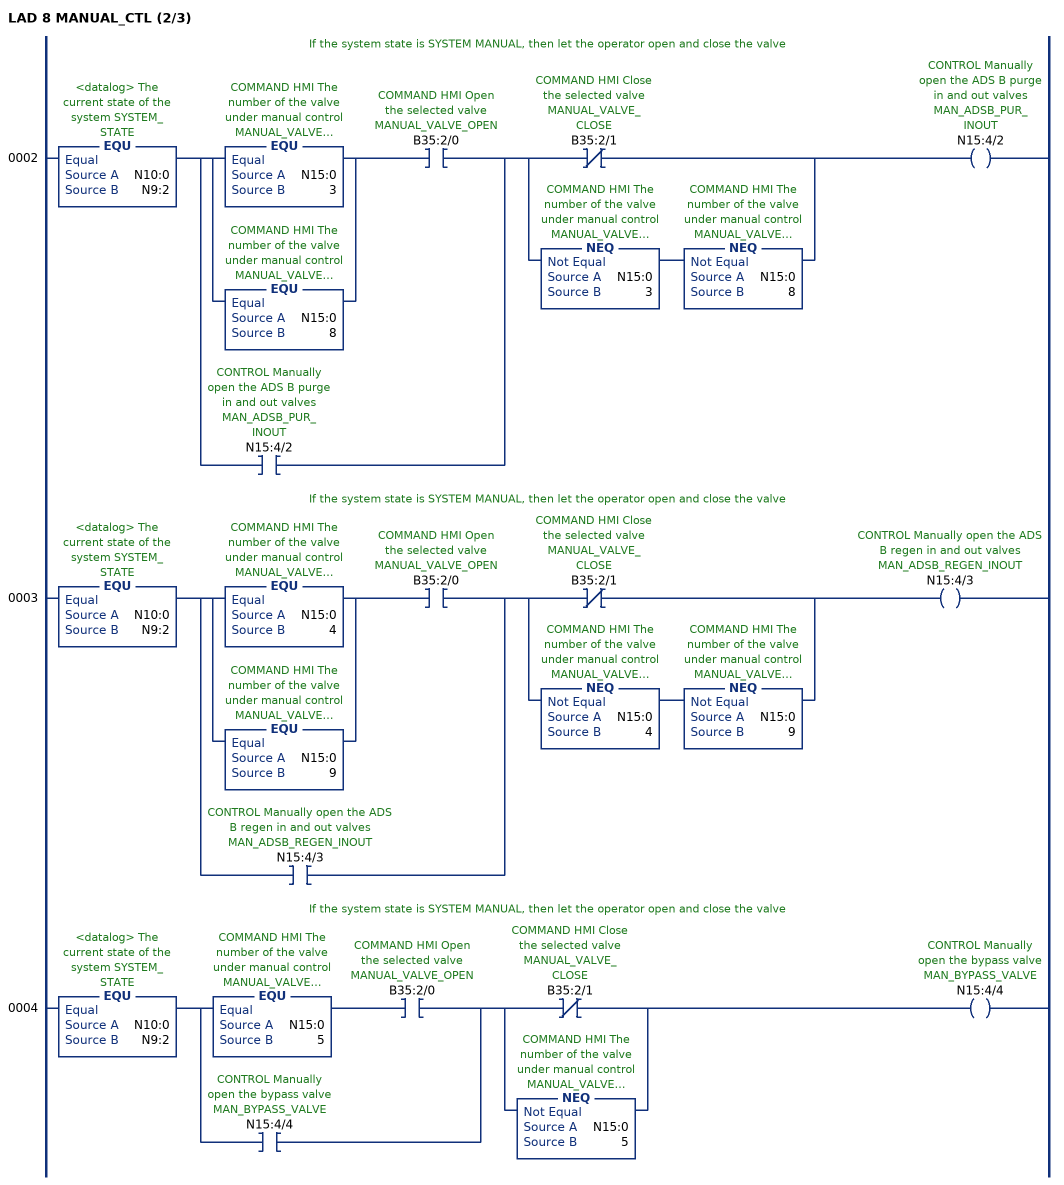
% Rung: 2 %
% If the system state is SYSTEM MANUAL, then let the operator open and close the valve %
SOR EQU N10:0 N9:2 BST BST EQU N15:0 3 NXB EQU N15:0 8 BND XIC B35:2/0 NXB XIC N15:4/2 BND BST XIO B35:2/1 NXB NEQ N15:0 3 NEQ N15:0 8 BND OTE N15:4/2 EOR
%   N10:0  SYSTEM_STATE  "<datalog> The current state of the system" %
%   N9:2  SYSTEM_MANUAL  "STATE System Manual" %
%   N15:0  MANUAL_VALVE_NUMBER  "COMMAND HMI The number of the valve under manual control" %
%   B35:2/0  MANUAL_VALVE_OPEN  "COMMAND HMI Open the selected valve" %
%   N15:4/2  MAN_ADSB_PUR_INOUT  "CONTROL Manually open the ADS B purge in and out valves" %
%   B35:2/1  MANUAL_VALVE_CLOSE  "COMMAND HMI Close the selected valve" %
% Rung: 3 %
% If the system state is SYSTEM MANUAL, then let the operator open and close the valve %
SOR EQU N10:0 N9:2 BST BST EQU N15:0 4 NXB EQU N15:0 9 BND XIC B35:2/0 NXB XIC N15:4/3 BND BST XIO B35:2/1 NXB NEQ N15:0 4 NEQ N15:0 9 BND OTE N15:4/3 EOR
%   N10:0  SYSTEM_STATE  "<datalog> The current state of the system" %
%   N9:2  SYSTEM_MANUAL  "STATE System Manual" %
%   N15:0  MANUAL_VALVE_NUMBER  "COMMAND HMI The number of the valve under manual control" %
%   B35:2/0  MANUAL_VALVE_OPEN  "COMMAND HMI Open the selected valve" %
%   N15:4/3  MAN_ADSB_REGEN_INOUT  "CONTROL Manually open the ADS B regen in and out valves" %
%   B35:2/1  MANUAL_VALVE_CLOSE  "COMMAND HMI Close the selected valve" %
% Rung: 4 %
% If the system state is SYSTEM MANUAL, then let the operator open and close the valve %
SOR EQU N10:0 N9:2 BST EQU N15:0 5 XIC B35:2/0 NXB XIC N15:4/4 BND BST XIO B35:2/1 NXB NEQ N15:0 5 BND OTE N15:4/4 EOR
%   N10:0  SYSTEM_STATE  "<datalog> The current state of the system" %
%   N9:2  SYSTEM_MANUAL  "STATE System Manual" %
%   N15:0  MANUAL_VALVE_NUMBER  "COMMAND HMI The number of the valve under manual control" %
%   B35:2/0  MANUAL_VALVE_OPEN  "COMMAND HMI Open the selected valve" %
%   N15:4/4  MAN_BYPASS_VALVE  "CONTROL Manually open the bypass valve" %
%   B35:2/1  MANUAL_VALVE_CLOSE  "COMMAND HMI Close the selected valve" %

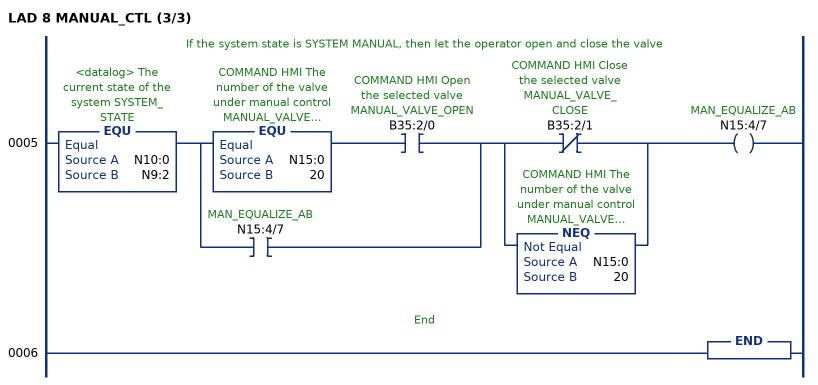
% Rung: 5 %
% If the system state is SYSTEM MANUAL, then let the operator open and close the valve %
SOR EQU N10:0 N9:2 BST EQU N15:0 20 XIC B35:2/0 NXB XIC N15:4/7 BND BST XIO B35:2/1 NXB NEQ N15:0 20 BND OTE N15:4/7 EOR
%   N10:0  SYSTEM_STATE  "<datalog> The current state of the system" %
%   N9:2  SYSTEM_MANUAL  "STATE System Manual" %
%   N15:0  MANUAL_VALVE_NUMBER  "COMMAND HMI The number of the valve under manual control" %
%   B35:2/0  MANUAL_VALVE_OPEN  "COMMAND HMI Open the selected valve" %
%   N15:4/7  MAN_EQUALIZE_AB %
%   B35:2/1  MANUAL_VALVE_CLOSE  "COMMAND HMI Close the selected valve" %
% Rung: 6 %
% End %
SOR END EOR

LADDER 10 "PURIFY"    % Operates the purify control %
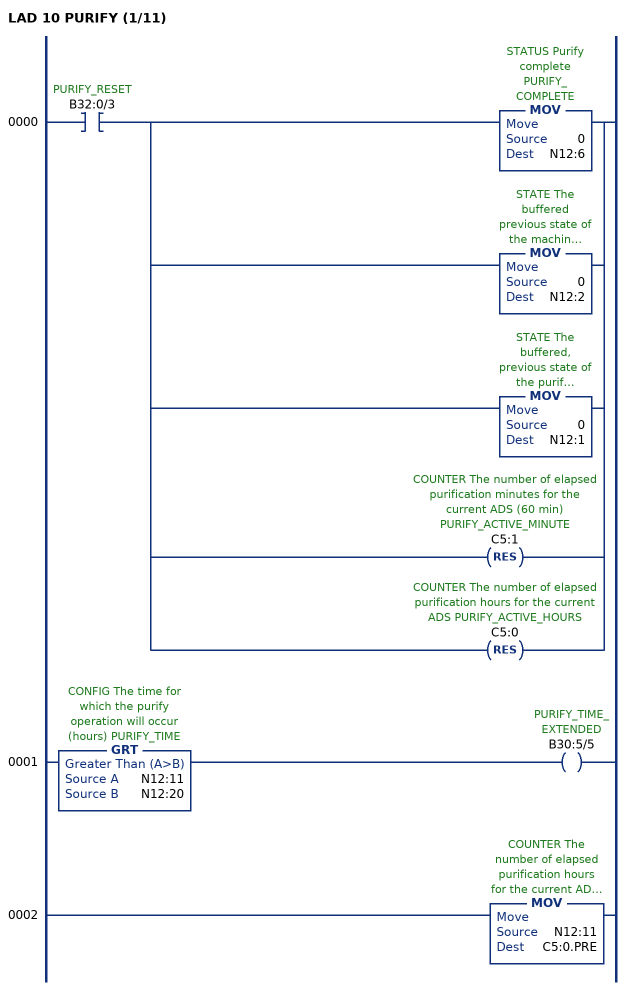
% Rung: 0 %
SOR XIC B32:0/3 BST MOV 0 N12:6 NXB MOV 0 N12:2 NXB MOV 0 N12:1 NXB RES C5:1 NXB RES C5:0 BND EOR
%   B32:0/3  PURIFY_RESET %
%   N12:6  PURIFY_COMPLETE  "STATUS Purify complete" %
%   N12:2  PURIFY_ALARM_BUFFER  "STATE The buffered previous state of the machine when the system alarm occured" %
%   N12:1  PURIFY_STDBY_BUFFER  "STATE The buffered, previous state of the purify process" %
%   C5:1  PURIFY_ACTIVE_MINUTE  "COUNTER The number of elapsed purification minutes for the current ADS (60 min)" %
%   C5:0  PURIFY_ACTIVE_HOURS  "COUNTER The number of elapsed purification hours for the current ADS" %
% Rung: 1 %
SOR GRT N12:11 N12:20 OTE B30:5/5 EOR
%   N12:11  PURIFY_TIME  "CONFIG The time for which the purify operation will occur (hours)" %
%   N12:20  DEFAULT_PURIFY_TIME %
%   B30:5/5  PURIFY_TIME_EXTENDED %
% Rung: 2 %
SOR MOV N12:11 C5:0.PRE EOR
%   N12:11  PURIFY_TIME  "CONFIG The time for which the purify operation will occur (hours)" %
%   C5:0  PURIFY_ACTIVE_HOURS  "COUNTER The number of elapsed purification hours for the current ADS" %

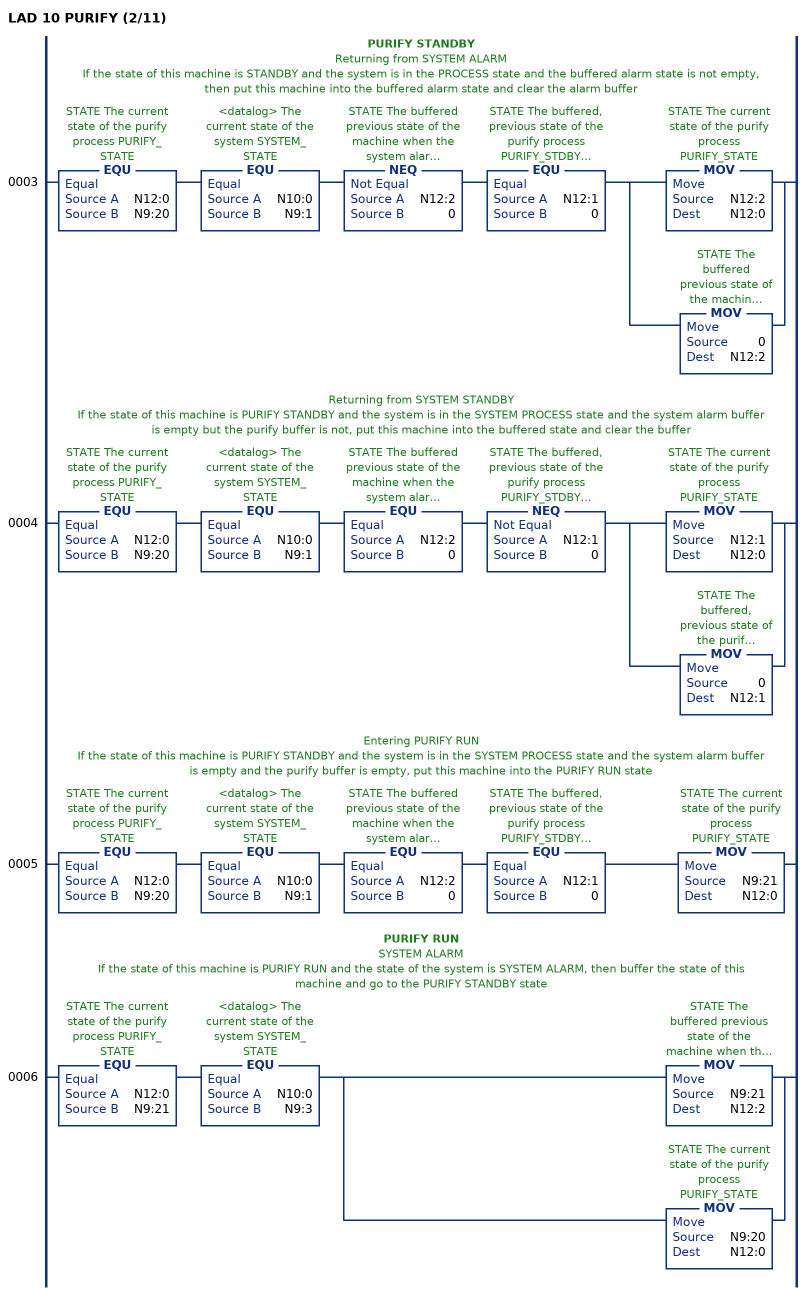
% Rung: 3 %
% TITLE: PURIFY STANDBY %
% Returning from SYSTEM ALARM
% If the state of this machine is STANDBY and the system is in the PROCESS state and the buffered alarm state is not empty, then put this machine into the buffered alarm state and clear the alarm buffer %
SOR EQU N12:0 N9:20 EQU N10:0 N9:1 NEQ N12:2 0 EQU N12:1 0 BST MOV N12:2 N12:0 NXB MOV 0 N12:2 BND EOR
%   N12:0  PURIFY_STATE  "STATE The current state of the purify process" %
%   N9:20  PURIFY_STANDBY  "STATE Purify Standby" %
%   N10:0  SYSTEM_STATE  "<datalog> The current state of the system" %
%   N9:1  SYSTEM_PROCESS  "STATE System Process" %
%   N12:2  PURIFY_ALARM_BUFFER  "STATE The buffered previous state of the machine when the system alarm occured" %
%   N12:1  PURIFY_STDBY_BUFFER  "STATE The buffered, previous state of the purify process" %
% Rung: 4 %
% Returning from SYSTEM STANDBY
% If the state of this machine is PURIFY STANDBY and the system is in the SYSTEM PROCESS state and the system alarm buffer is empty but the purify buffer is not, put this machine into the buffered state and clear the buffer %
SOR EQU N12:0 N9:20 EQU N10:0 N9:1 EQU N12:2 0 NEQ N12:1 0 BST MOV N12:1 N12:0 NXB MOV 0 N12:1 BND EOR
%   N12:0  PURIFY_STATE  "STATE The current state of the purify process" %
%   N9:20  PURIFY_STANDBY  "STATE Purify Standby" %
%   N10:0  SYSTEM_STATE  "<datalog> The current state of the system" %
%   N9:1  SYSTEM_PROCESS  "STATE System Process" %
%   N12:2  PURIFY_ALARM_BUFFER  "STATE The buffered previous state of the machine when the system alarm occured" %
%   N12:1  PURIFY_STDBY_BUFFER  "STATE The buffered, previous state of the purify process" %
% Rung: 5 %
% Entering PURIFY RUN
% If the state of this machine is PURIFY STANDBY and the system is in the SYSTEM PROCESS state and the system alarm buffer is empty and the purify buffer is empty, put this machine into the PURIFY RUN state %
SOR EQU N12:0 N9:20 EQU N10:0 N9:1 EQU N12:2 0 EQU N12:1 0 MOV N9:21 N12:0 EOR
%   N12:0  PURIFY_STATE  "STATE The current state of the purify process" %
%   N9:20  PURIFY_STANDBY  "STATE Purify Standby" %
%   N10:0  SYSTEM_STATE  "<datalog> The current state of the system" %
%   N9:1  SYSTEM_PROCESS  "STATE System Process" %
%   N12:2  PURIFY_ALARM_BUFFER  "STATE The buffered previous state of the machine when the system alarm occured" %
%   N12:1  PURIFY_STDBY_BUFFER  "STATE The buffered, previous state of the purify process" %
%   N9:21  PURIFY_RUN  "STATE Purify running" %
% Rung: 6 %
% TITLE: PURIFY RUN %
% SYSTEM ALARM
% If the state of this machine is PURIFY RUN and the state of the system is SYSTEM ALARM, then buffer the state of this machine and go to the PURIFY STANDBY state %
SOR EQU N12:0 N9:21 EQU N10:0 N9:3 BST MOV N9:21 N12:2 NXB MOV N9:20 N12:0 BND EOR
%   N12:0  PURIFY_STATE  "STATE The current state of the purify process" %
%   N9:21  PURIFY_RUN  "STATE Purify running" %
%   N10:0  SYSTEM_STATE  "<datalog> The current state of the system" %
%   N9:3  SYSTEM_ALARM  "STATE System Alarm" %
%   N12:2  PURIFY_ALARM_BUFFER  "STATE The buffered previous state of the machine when the system alarm occured" %
%   N9:20  PURIFY_STANDBY  "STATE Purify Standby" %

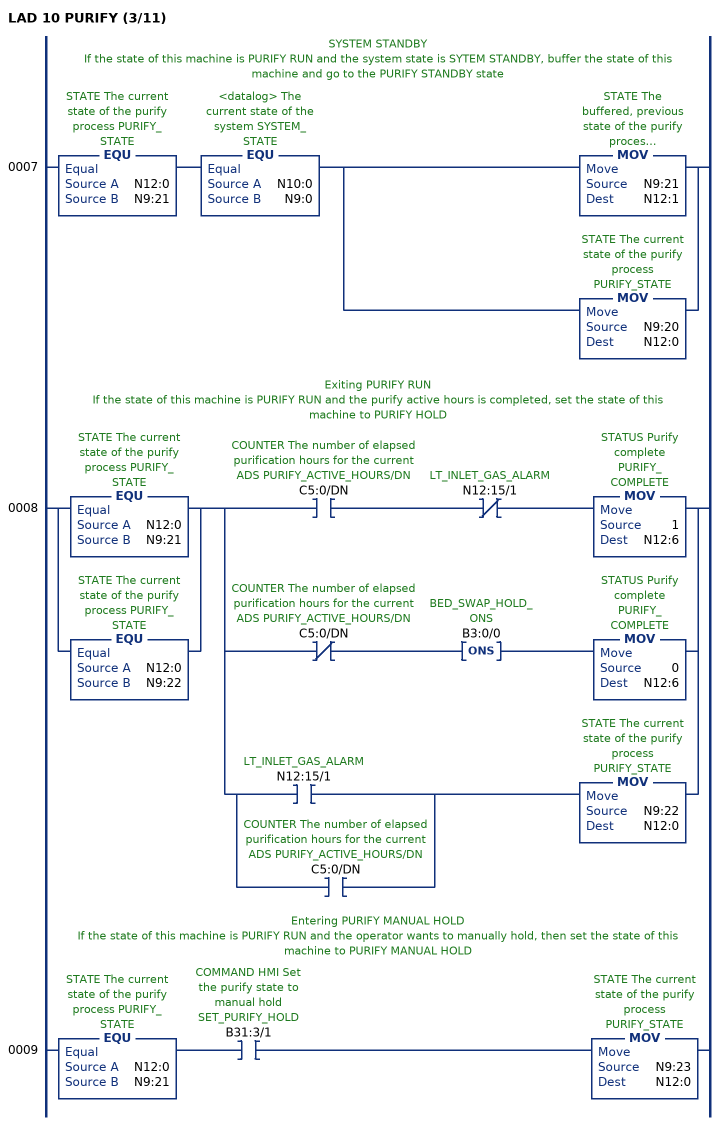
% Rung: 7 %
% SYSTEM STANDBY
% If the state of this machine is PURIFY RUN and the system state is SYTEM STANDBY, buffer the state of this machine and go to the PURIFY STANDBY state %
SOR EQU N12:0 N9:21 EQU N10:0 N9:0 BST MOV N9:21 N12:1 NXB MOV N9:20 N12:0 BND EOR
%   N12:0  PURIFY_STATE  "STATE The current state of the purify process" %
%   N9:21  PURIFY_RUN  "STATE Purify running" %
%   N10:0  SYSTEM_STATE  "<datalog> The current state of the system" %
%   N9:0  SYSTEM_STANDBY  "STATE System Standby" %
%   N12:1  PURIFY_STDBY_BUFFER  "STATE The buffered, previous state of the purify process" %
%   N9:20  PURIFY_STANDBY  "STATE Purify Standby" %
% Rung: 8 %
% Exiting PURIFY RUN
% If the state of this machine is PURIFY RUN and the purify active hours is completed, set the state of this machine to PURIFY HOLD %
SOR BST EQU N12:0 N9:21 NXB EQU N12:0 N9:22 BND BST XIC C5:0/DN XIO N12:15/1 MOV 1 N12:6 NXB XIO C5:0/DN ONS B3:0/0 MOV 0 N12:6 NXB BST XIC N12:15/1 NXB XIC C5:0/DN BND MOV N9:22 N12:0 BND EOR
%   N12:0  PURIFY_STATE  "STATE The current state of the purify process" %
%   N9:21  PURIFY_RUN  "STATE Purify running" %
%   N9:22  PURIFY_HOLD  "STATE Purify Hold" %
%   C5:0  PURIFY_ACTIVE_HOURS  "COUNTER The number of elapsed purification hours for the current ADS" %
%   N12:15/1  LT_INLET_GAS_ALARM %
%   N12:6  PURIFY_COMPLETE  "STATUS Purify complete" %
%   B3:0/0  BED_SWAP_HOLD_ONS %
% Rung: 9 %
% Entering PURIFY MANUAL HOLD
% If the state of this machine is PURIFY RUN and the operator wants to manually hold, then set the state of this machine to PURIFY MANUAL HOLD %
SOR EQU N12:0 N9:21 XIC B31:3/1 MOV N9:23 N12:0 EOR
%   N12:0  PURIFY_STATE  "STATE The current state of the purify process" %
%   N9:21  PURIFY_RUN  "STATE Purify running" %
%   B31:3/1  SET_PURIFY_HOLD  "COMMAND HMI Set the purify state to manual hold" %
%   N9:23  PURIFY_MANUAL_HOLD  "STATE Purify Manual Hold" %

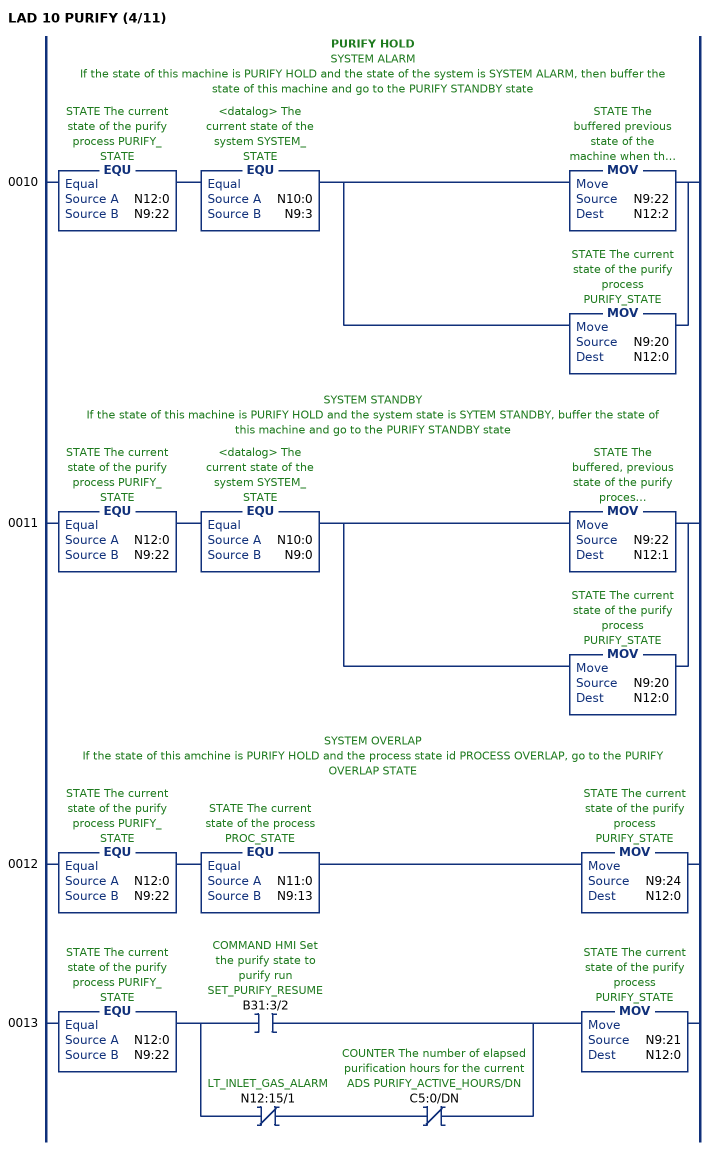
% Rung: 10 %
% TITLE: PURIFY HOLD %
% SYSTEM ALARM
% If the state of this machine is PURIFY HOLD and the state of the system is SYSTEM ALARM, then buffer the state of this machine and go to the PURIFY STANDBY state %
SOR EQU N12:0 N9:22 EQU N10:0 N9:3 BST MOV N9:22 N12:2 NXB MOV N9:20 N12:0 BND EOR
%   N12:0  PURIFY_STATE  "STATE The current state of the purify process" %
%   N9:22  PURIFY_HOLD  "STATE Purify Hold" %
%   N10:0  SYSTEM_STATE  "<datalog> The current state of the system" %
%   N9:3  SYSTEM_ALARM  "STATE System Alarm" %
%   N12:2  PURIFY_ALARM_BUFFER  "STATE The buffered previous state of the machine when the system alarm occured" %
%   N9:20  PURIFY_STANDBY  "STATE Purify Standby" %
% Rung: 11 %
% SYSTEM STANDBY
% If the state of this machine is PURIFY HOLD and the system state is SYTEM STANDBY, buffer the state of this machine and go to the PURIFY STANDBY state %
SOR EQU N12:0 N9:22 EQU N10:0 N9:0 BST MOV N9:22 N12:1 NXB MOV N9:20 N12:0 BND EOR
%   N12:0  PURIFY_STATE  "STATE The current state of the purify process" %
%   N9:22  PURIFY_HOLD  "STATE Purify Hold" %
%   N10:0  SYSTEM_STATE  "<datalog> The current state of the system" %
%   N9:0  SYSTEM_STANDBY  "STATE System Standby" %
%   N12:1  PURIFY_STDBY_BUFFER  "STATE The buffered, previous state of the purify process" %
%   N9:20  PURIFY_STANDBY  "STATE Purify Standby" %
% Rung: 12 %
% SYSTEM OVERLAP
% If the state of this amchine is PURIFY HOLD and the process state id PROCESS OVERLAP, go to the PURIFY OVERLAP STATE %
SOR EQU N12:0 N9:22 EQU N11:0 N9:13 MOV N9:24 N12:0 EOR
%   N12:0  PURIFY_STATE  "STATE The current state of the purify process" %
%   N9:22  PURIFY_HOLD  "STATE Purify Hold" %
%   N11:0  PROC_STATE  "STATE The current state of the process" %
%   N9:13  PROC_OVERLAP  "STATE Process Purify Overlap" %
%   N9:24  PURIFY_OVERLAP  "STATE Puriify Overlap" %
% Rung: 13 %
SOR EQU N12:0 N9:22 BST XIC B31:3/2 NXB XIO N12:15/1 XIO C5:0/DN BND MOV N9:21 N12:0 EOR
%   N12:0  PURIFY_STATE  "STATE The current state of the purify process" %
%   N9:22  PURIFY_HOLD  "STATE Purify Hold" %
%   B31:3/2  SET_PURIFY_RESUME  "COMMAND HMI Set the purify state to purify run" %
%   N12:15/1  LT_INLET_GAS_ALARM %
%   C5:0  PURIFY_ACTIVE_HOURS  "COUNTER The number of elapsed purification hours for the current ADS" %
%   N9:21  PURIFY_RUN  "STATE Purify running" %

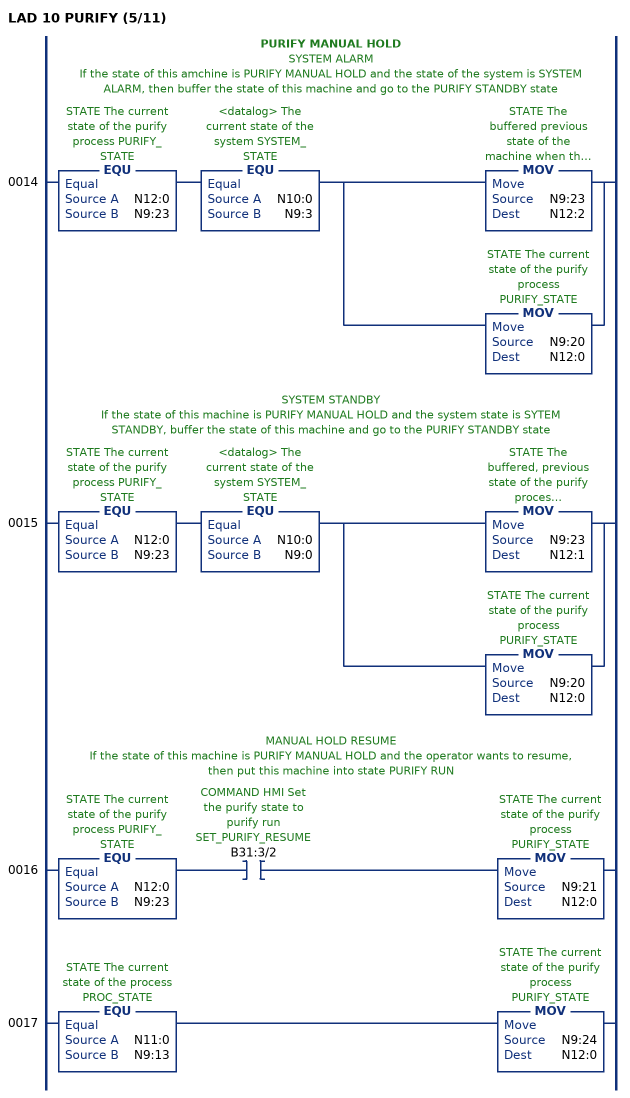
% Rung: 14 %
% TITLE: PURIFY MANUAL HOLD %
% SYSTEM ALARM
% If the state of this amchine is PURIFY MANUAL HOLD and the state of the system is SYSTEM ALARM, then buffer the state of this machine and go to the PURIFY STANDBY state %
SOR EQU N12:0 N9:23 EQU N10:0 N9:3 BST MOV N9:23 N12:2 NXB MOV N9:20 N12:0 BND EOR
%   N12:0  PURIFY_STATE  "STATE The current state of the purify process" %
%   N9:23  PURIFY_MANUAL_HOLD  "STATE Purify Manual Hold" %
%   N10:0  SYSTEM_STATE  "<datalog> The current state of the system" %
%   N9:3  SYSTEM_ALARM  "STATE System Alarm" %
%   N12:2  PURIFY_ALARM_BUFFER  "STATE The buffered previous state of the machine when the system alarm occured" %
%   N9:20  PURIFY_STANDBY  "STATE Purify Standby" %
% Rung: 15 %
% SYSTEM STANDBY
% If the state of this machine is PURIFY MANUAL HOLD and the system state is SYTEM STANDBY, buffer the state of this machine and go to the PURIFY STANDBY state %
SOR EQU N12:0 N9:23 EQU N10:0 N9:0 BST MOV N9:23 N12:1 NXB MOV N9:20 N12:0 BND EOR
%   N12:0  PURIFY_STATE  "STATE The current state of the purify process" %
%   N9:23  PURIFY_MANUAL_HOLD  "STATE Purify Manual Hold" %
%   N10:0  SYSTEM_STATE  "<datalog> The current state of the system" %
%   N9:0  SYSTEM_STANDBY  "STATE System Standby" %
%   N12:1  PURIFY_STDBY_BUFFER  "STATE The buffered, previous state of the purify process" %
%   N9:20  PURIFY_STANDBY  "STATE Purify Standby" %
% Rung: 16 %
% MANUAL HOLD RESUME
% If the state of this machine is PURIFY MANUAL HOLD and the operator wants to resume, then put this machine into state PURIFY RUN %
SOR EQU N12:0 N9:23 XIC B31:3/2 MOV N9:21 N12:0 EOR
%   N12:0  PURIFY_STATE  "STATE The current state of the purify process" %
%   N9:23  PURIFY_MANUAL_HOLD  "STATE Purify Manual Hold" %
%   B31:3/2  SET_PURIFY_RESUME  "COMMAND HMI Set the purify state to purify run" %
%   N9:21  PURIFY_RUN  "STATE Purify running" %
% Rung: 17 %
SOR EQU N11:0 N9:13 MOV N9:24 N12:0 EOR
%   N11:0  PROC_STATE  "STATE The current state of the process" %
%   N9:13  PROC_OVERLAP  "STATE Process Purify Overlap" %
%   N9:24  PURIFY_OVERLAP  "STATE Puriify Overlap" %
%   N12:0  PURIFY_STATE  "STATE The current state of the purify process" %

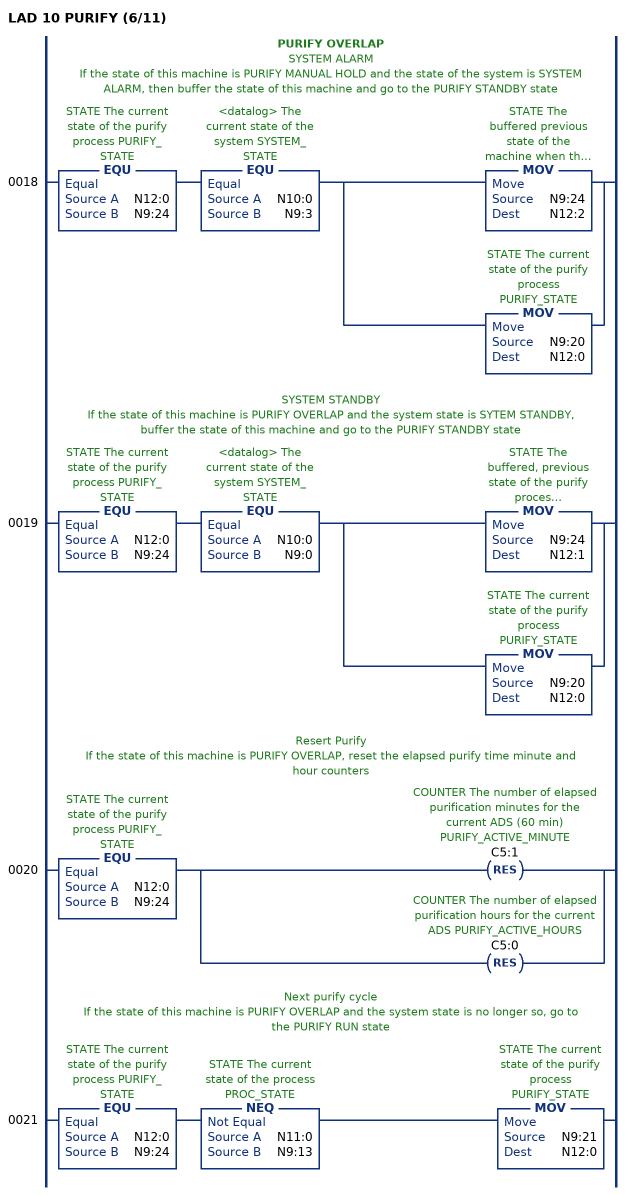
% Rung: 18 %
% TITLE: PURIFY OVERLAP %
% SYSTEM ALARM
% If the state of this machine is PURIFY MANUAL HOLD and the state of the system is SYSTEM ALARM, then buffer the state of this machine and go to the PURIFY STANDBY state %
SOR EQU N12:0 N9:24 EQU N10:0 N9:3 BST MOV N9:24 N12:2 NXB MOV N9:20 N12:0 BND EOR
%   N12:0  PURIFY_STATE  "STATE The current state of the purify process" %
%   N9:24  PURIFY_OVERLAP  "STATE Puriify Overlap" %
%   N10:0  SYSTEM_STATE  "<datalog> The current state of the system" %
%   N9:3  SYSTEM_ALARM  "STATE System Alarm" %
%   N12:2  PURIFY_ALARM_BUFFER  "STATE The buffered previous state of the machine when the system alarm occured" %
%   N9:20  PURIFY_STANDBY  "STATE Purify Standby" %
% Rung: 19 %
% SYSTEM STANDBY
% If the state of this machine is PURIFY OVERLAP and the system state is SYTEM STANDBY, buffer the state of this machine and go to the PURIFY STANDBY state %
SOR EQU N12:0 N9:24 EQU N10:0 N9:0 BST MOV N9:24 N12:1 NXB MOV N9:20 N12:0 BND EOR
%   N12:0  PURIFY_STATE  "STATE The current state of the purify process" %
%   N9:24  PURIFY_OVERLAP  "STATE Puriify Overlap" %
%   N10:0  SYSTEM_STATE  "<datalog> The current state of the system" %
%   N9:0  SYSTEM_STANDBY  "STATE System Standby" %
%   N12:1  PURIFY_STDBY_BUFFER  "STATE The buffered, previous state of the purify process" %
%   N9:20  PURIFY_STANDBY  "STATE Purify Standby" %
% Rung: 20 %
% Resert Purify
% If the state of this machine is PURIFY OVERLAP, reset the elapsed purify time minute and hour counters %
SOR EQU N12:0 N9:24 BST RES C5:1 NXB RES C5:0 BND EOR
%   N12:0  PURIFY_STATE  "STATE The current state of the purify process" %
%   N9:24  PURIFY_OVERLAP  "STATE Puriify Overlap" %
%   C5:1  PURIFY_ACTIVE_MINUTE  "COUNTER The number of elapsed purification minutes for the current ADS (60 min)" %
%   C5:0  PURIFY_ACTIVE_HOURS  "COUNTER The number of elapsed purification hours for the current ADS" %
% Rung: 21 %
% Next purify cycle
% If the state of this machine is PURIFY OVERLAP and the system state is no longer so, go to the PURIFY RUN state %
SOR EQU N12:0 N9:24 NEQ N11:0 N9:13 MOV N9:21 N12:0 EOR
%   N12:0  PURIFY_STATE  "STATE The current state of the purify process" %
%   N9:24  PURIFY_OVERLAP  "STATE Puriify Overlap" %
%   N11:0  PROC_STATE  "STATE The current state of the process" %
%   N9:13  PROC_OVERLAP  "STATE Process Purify Overlap" %
%   N9:21  PURIFY_RUN  "STATE Purify running" %

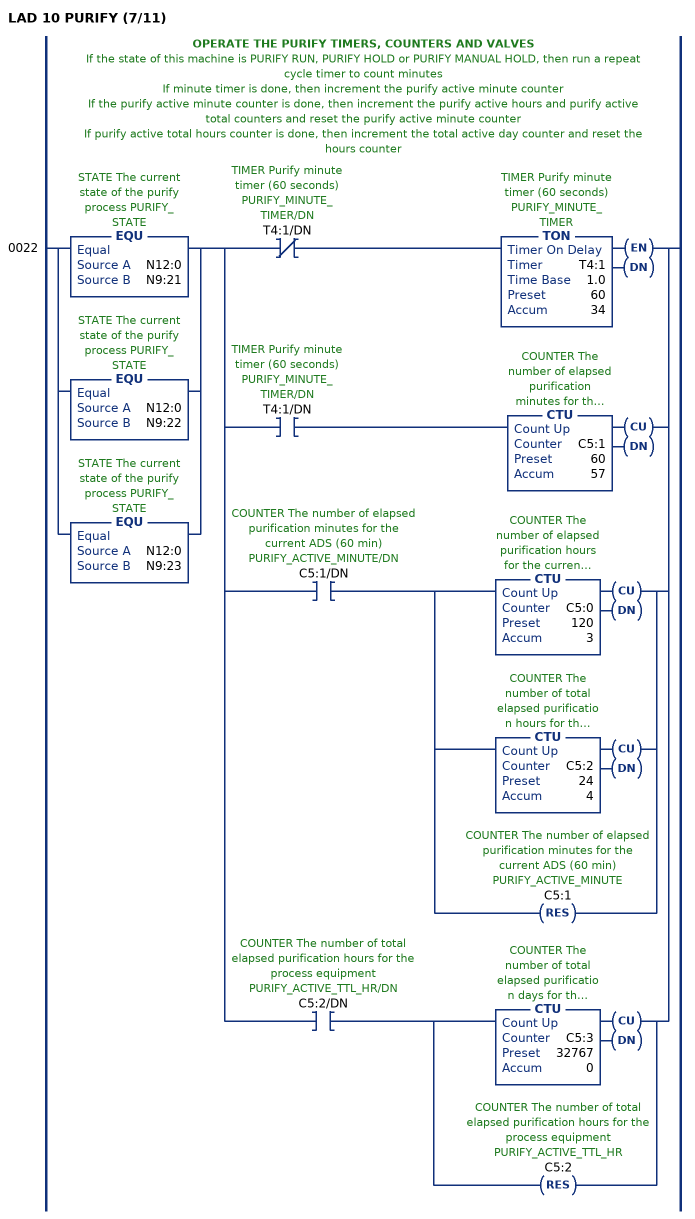
% Rung: 22 %
% TITLE: OPERATE THE PURIFY TIMERS, COUNTERS AND VALVES %
% If the state of this machine is PURIFY RUN, PURIFY HOLD or PURIFY MANUAL HOLD, then run a repeat cycle timer to count minutes
% If minute timer is done, then increment the purify active minute counter
% If the purify active minute counter is done, then increment the purify active hours and purify active total counters and reset the purify active minute counter
% If purify active total hours counter is done, then increment the total active day counter and reset the hours counter %
SOR BST EQU N12:0 N9:21 NXB EQU N12:0 N9:22 NXB EQU N12:0 N9:23 BND BST XIO T4:1/DN TON T4:1 1.0 60 34 NXB XIC T4:1/DN CTU C5:1 60 57 NXB XIC C5:1/DN BST CTU C5:0 120 3 NXB CTU C5:2 24 4 NXB RES C5:1 BND NXB XIC C5:2/DN BST CTU C5:3 32767 0 NXB RES C5:2 BND BND EOR
%   N12:0  PURIFY_STATE  "STATE The current state of the purify process" %
%   N9:21  PURIFY_RUN  "STATE Purify running" %
%   N9:22  PURIFY_HOLD  "STATE Purify Hold" %
%   N9:23  PURIFY_MANUAL_HOLD  "STATE Purify Manual Hold" %
%   T4:1  PURIFY_MINUTE_TIMER  "TIMER Purify minute timer (60 seconds)" %
%   C5:1  PURIFY_ACTIVE_MINUTE  "COUNTER The number of elapsed purification minutes for the current ADS (60 min)" %
%   C5:0  PURIFY_ACTIVE_HOURS  "COUNTER The number of elapsed purification hours for the current ADS" %
%   C5:2  PURIFY_ACTIVE_TTL_HR  "COUNTER The number of total elapsed purification hours for the process equipment" %
%   C5:3  PURIFY_ACTIVE_TTL_DY  "COUNTER The number of total elapsed purification days for the process equipment" %

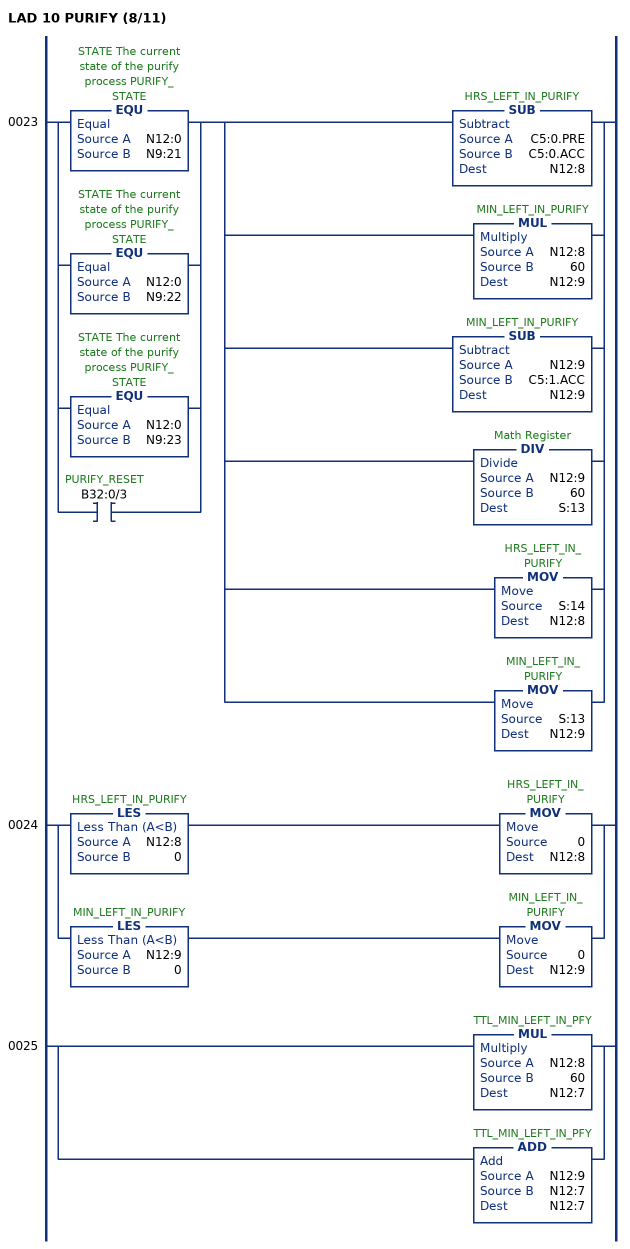
% Rung: 23 %
SOR BST EQU N12:0 N9:21 NXB EQU N12:0 N9:22 NXB EQU N12:0 N9:23 NXB XIC B32:0/3 BND BST SUB C5:0.PRE C5:0.ACC N12:8 NXB MUL N12:8 60 N12:9 NXB SUB N12:9 C5:1.ACC N12:9 NXB DIV N12:9 60 S:13 NXB MOV S:14 N12:8 NXB MOV S:13 N12:9 BND EOR
%   N12:0  PURIFY_STATE  "STATE The current state of the purify process" %
%   N9:21  PURIFY_RUN  "STATE Purify running" %
%   N9:22  PURIFY_HOLD  "STATE Purify Hold" %
%   N9:23  PURIFY_MANUAL_HOLD  "STATE Purify Manual Hold" %
%   B32:0/3  PURIFY_RESET %
%   C5:0  PURIFY_ACTIVE_HOURS  "COUNTER The number of elapsed purification hours for the current ADS" %
%   N12:8  HRS_LEFT_IN_PURIFY %
%   N12:9  MIN_LEFT_IN_PURIFY %
%   C5:1  PURIFY_ACTIVE_MINUTE  "COUNTER The number of elapsed purification minutes for the current ADS (60 min)" %
%   S:13  "Math Register" %
%   S:14  "Math Register" %
% Rung: 24 %
SOR BST LES N12:8 0 MOV 0 N12:8 NXB LES N12:9 0 MOV 0 N12:9 BND EOR
%   N12:8  HRS_LEFT_IN_PURIFY %
%   N12:9  MIN_LEFT_IN_PURIFY %
% Rung: 25 %
SOR BST MUL N12:8 60 N12:7 NXB ADD N12:9 N12:7 N12:7 BND EOR
%   N12:8  HRS_LEFT_IN_PURIFY %
%   N12:7  TTL_MIN_LEFT_IN_PFY %
%   N12:9  MIN_LEFT_IN_PURIFY %

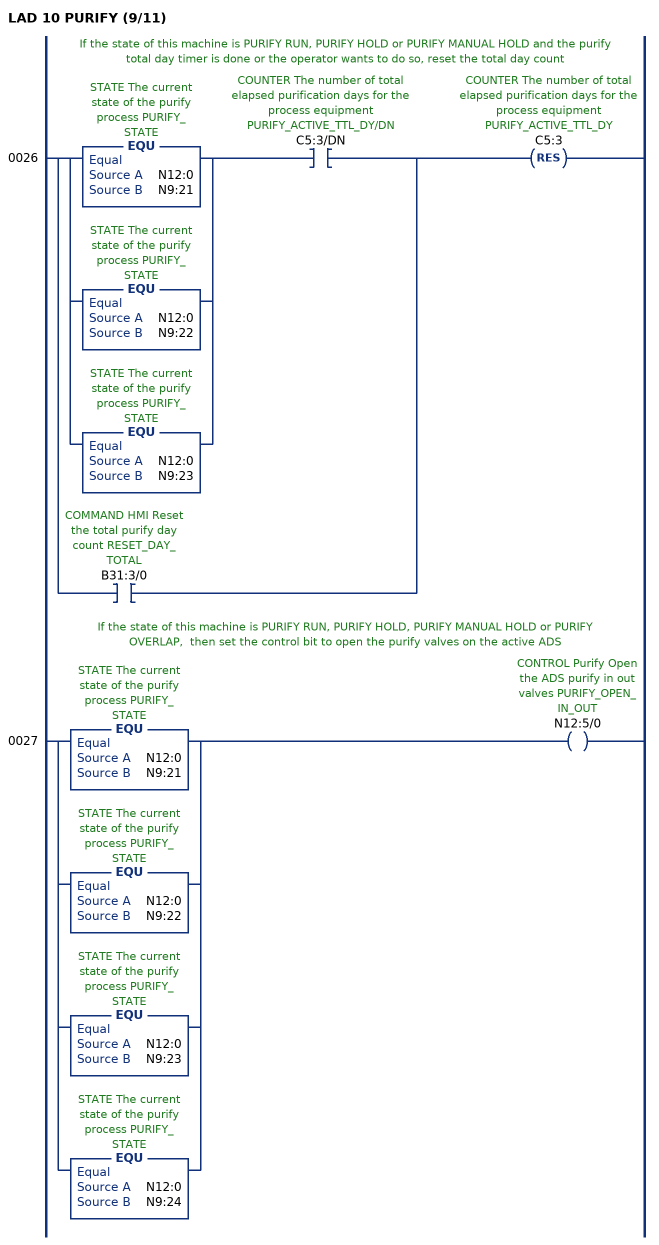
% Rung: 26 %
% If the state of this machine is PURIFY RUN, PURIFY HOLD or PURIFY MANUAL HOLD and the purify total day timer is done or the operator wants to do so, reset the total day count %
SOR BST BST EQU N12:0 N9:21 NXB EQU N12:0 N9:22 NXB EQU N12:0 N9:23 BND XIC C5:3/DN NXB XIC B31:3/0 BND RES C5:3 EOR
%   N12:0  PURIFY_STATE  "STATE The current state of the purify process" %
%   N9:21  PURIFY_RUN  "STATE Purify running" %
%   N9:22  PURIFY_HOLD  "STATE Purify Hold" %
%   N9:23  PURIFY_MANUAL_HOLD  "STATE Purify Manual Hold" %
%   C5:3  PURIFY_ACTIVE_TTL_DY  "COUNTER The number of total elapsed purification days for the process equipment" %
%   B31:3/0  RESET_DAY_TOTAL  "COMMAND HMI Reset the total purify day count" %
% Rung: 27 %
% If the state of this machine is PURIFY RUN, PURIFY HOLD, PURIFY MANUAL HOLD or PURIFY OVERLAP,  then set the control bit to open the purify valves on the active ADS %
SOR BST EQU N12:0 N9:21 NXB EQU N12:0 N9:22 NXB EQU N12:0 N9:23 NXB EQU N12:0 N9:24 BND OTE N12:5/0 EOR
%   N12:0  PURIFY_STATE  "STATE The current state of the purify process" %
%   N9:21  PURIFY_RUN  "STATE Purify running" %
%   N9:22  PURIFY_HOLD  "STATE Purify Hold" %
%   N9:23  PURIFY_MANUAL_HOLD  "STATE Purify Manual Hold" %
%   N9:24  PURIFY_OVERLAP  "STATE Puriify Overlap" %
%   N12:5/0  PURIFY_OPEN_IN_OUT  "CONTROL Purify Open the ADS purify in out valves" %

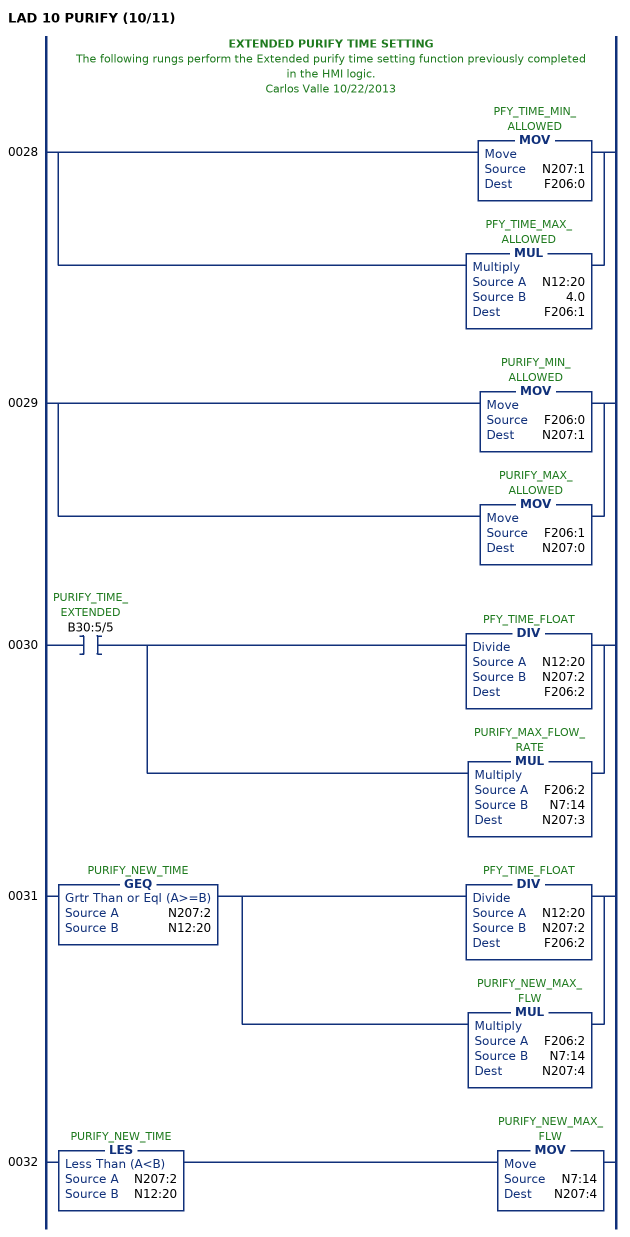
% Rung: 28 %
% TITLE: EXTENDED PURIFY TIME SETTING %
% The following rungs perform the Extended purify time setting function previously completed in the HMI logic.
% Carlos Valle 10/22/2013 %
SOR BST MOV N207:1 F206:0 NXB MUL N12:20 4.0 F206:1 BND EOR
%   N207:1  PURIFY_MIN_ALLOWED %
%   F206:0  PFY_TIME_MIN_ALLOWED %
%   N12:20  DEFAULT_PURIFY_TIME %
%   F206:1  PFY_TIME_MAX_ALLOWED %
% Rung: 29 %
SOR BST MOV F206:0 N207:1 NXB MOV F206:1 N207:0 BND EOR
%   F206:0  PFY_TIME_MIN_ALLOWED %
%   N207:1  PURIFY_MIN_ALLOWED %
%   F206:1  PFY_TIME_MAX_ALLOWED %
%   N207:0  PURIFY_MAX_ALLOWED %
% Rung: 30 %
SOR XIC B30:5/5 BST DIV N12:20 N207:2 F206:2 NXB MUL F206:2 N7:14 N207:3 BND EOR
%   B30:5/5  PURIFY_TIME_EXTENDED %
%   N12:20  DEFAULT_PURIFY_TIME %
%   N207:2  PURIFY_NEW_TIME %
%   F206:2  PFY_TIME_FLOAT %
%   N7:14  PURIFIER_SIZE %
%   N207:3  PURIFY_MAX_FLOW_RATE %
% Rung: 31 %
SOR GEQ N207:2 N12:20 BST DIV N12:20 N207:2 F206:2 NXB MUL F206:2 N7:14 N207:4 BND EOR
%   N207:2  PURIFY_NEW_TIME %
%   N12:20  DEFAULT_PURIFY_TIME %
%   F206:2  PFY_TIME_FLOAT %
%   N7:14  PURIFIER_SIZE %
%   N207:4  PURIFY_NEW_MAX_FLW %
% Rung: 32 %
SOR LES N207:2 N12:20 MOV N7:14 N207:4 EOR
%   N207:2  PURIFY_NEW_TIME %
%   N12:20  DEFAULT_PURIFY_TIME %
%   N7:14  PURIFIER_SIZE %
%   N207:4  PURIFY_NEW_MAX_FLW %

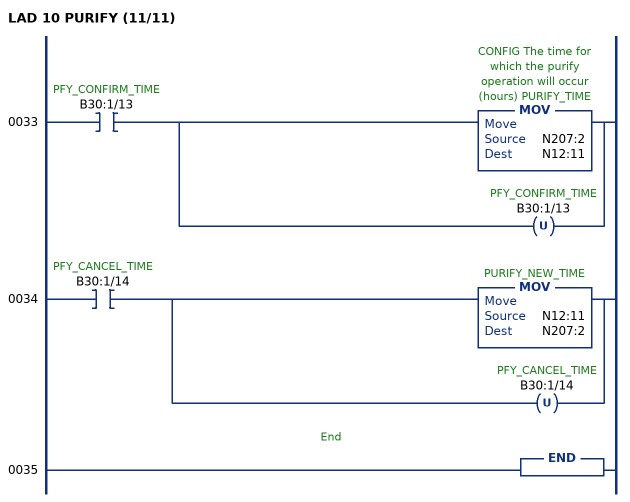
% Rung: 33 %
SOR XIC B30:1/13 BST MOV N207:2 N12:11 NXB OTU B30:1/13 BND EOR
%   B30:1/13  PFY_CONFIRM_TIME %
%   N207:2  PURIFY_NEW_TIME %
%   N12:11  PURIFY_TIME  "CONFIG The time for which the purify operation will occur (hours)" %
% Rung: 34 %
SOR XIC B30:1/14 BST MOV N12:11 N207:2 NXB OTU B30:1/14 BND EOR
%   B30:1/14  PFY_CANCEL_TIME %
%   N12:11  PURIFY_TIME  "CONFIG The time for which the purify operation will occur (hours)" %
%   N207:2  PURIFY_NEW_TIME %
% Rung: 35 %
% End %
SOR END EOR

LADDER 11 "REGEN"    % Operates the regen control %
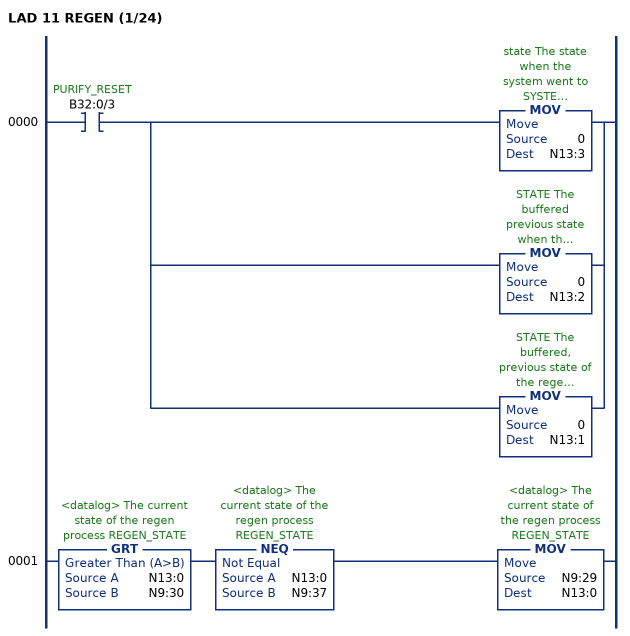
% Rung: 0 %
SOR XIC B32:0/3 BST MOV 0 N13:3 NXB MOV 0 N13:2 NXB MOV 0 N13:1 BND EOR
%   B32:0/3  PURIFY_RESET %
%   N13:3  REGEN_STANDBY_BUFFER  "state The state when the system went to SYSTEM STANDBY" %
%   N13:2  REGEN_ALARM_BUFFER  "STATE The buffered previous state when the system alarm occured" %
%   N13:1  REGEN_BUFFER  "STATE The buffered, previous state of the regen process" %
% Rung: 1 %
SOR GRT N13:0 N9:30 NEQ N13:0 N9:37 MOV N9:29 N13:0 EOR
%   N13:0  REGEN_STATE  "<datalog> The current state of the regen process" %
%   N9:30  REGEN_STANDBY  "STATE Regen Standby" %
%   N9:37  REGEN_ALARM  "STATE Regen Alarm" %
%   N9:29  REGEN_IDLE %

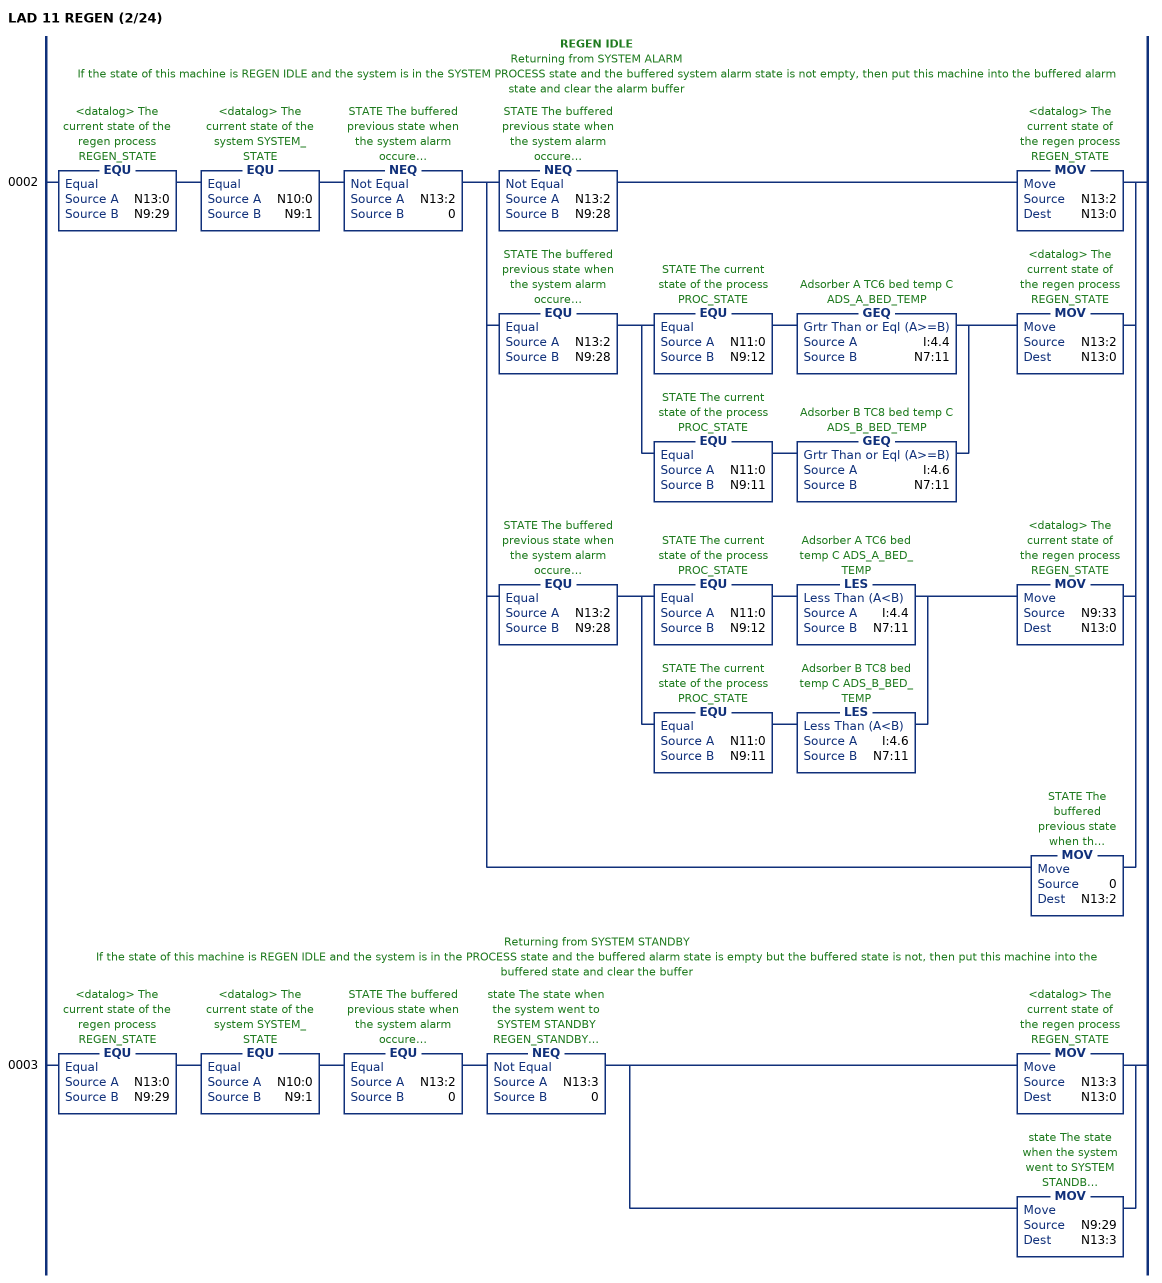
% Rung: 2 %
% TITLE: REGEN IDLE %
% Returning from SYSTEM ALARM
% If the state of this machine is REGEN IDLE and the system is in the SYSTEM PROCESS state and the buffered system alarm state is not empty, then put this machine into the buffered alarm state and clear the alarm buffer %
SOR EQU N13:0 N9:29 EQU N10:0 N9:1 NEQ N13:2 0 BST NEQ N13:2 N9:28 MOV N13:2 N13:0 NXB EQU N13:2 N9:28 BST EQU N11:0 N9:12 GEQ I:4.4 N7:11 NXB EQU N11:0 N9:11 GEQ I:4.6 N7:11 BND MOV N13:2 N13:0 NXB EQU N13:2 N9:28 BST EQU N11:0 N9:12 LES I:4.4 N7:11 NXB EQU N11:0 N9:11 LES I:4.6 N7:11 BND MOV N9:33 N13:0 NXB MOV 0 N13:2 BND EOR
%   N13:0  REGEN_STATE  "<datalog> The current state of the regen process" %
%   N9:29  REGEN_IDLE %
%   N10:0  SYSTEM_STATE  "<datalog> The current state of the system" %
%   N9:1  SYSTEM_PROCESS  "STATE System Process" %
%   N13:2  REGEN_ALARM_BUFFER  "STATE The buffered previous state when the system alarm occured" %
%   N9:28  REGEN_RUN %
%   N11:0  PROC_STATE  "STATE The current state of the process" %
%   N9:12  PROC_REGEN_A  "STATE Process Purify B" %
%   I:4.4  ADS_A_BED_TEMP  "Adsorber A TC6 bed temp C" %
%   N7:11  ADS_BED_TEMP_HIGH  "CONFIG The temp at which the regen process may continue" %
%   N9:11  PROC_REGEN_B  "STATE Process Purify A" %
%   I:4.6  ADS_B_BED_TEMP  "Adsorber B TC8 bed temp C" %
%   N9:33  REGEN_HEAT_BED  "STATE Regen Heat wall" %
% Rung: 3 %
% Returning from SYSTEM STANDBY
% If the state of this machine is REGEN IDLE and the system is in the PROCESS state and the buffered alarm state is empty but the buffered state is not, then put this machine into the buffered state and clear the buffer %
SOR EQU N13:0 N9:29 EQU N10:0 N9:1 EQU N13:2 0 NEQ N13:3 0 BST MOV N13:3 N13:0 NXB MOV N9:29 N13:3 BND EOR
%   N13:0  REGEN_STATE  "<datalog> The current state of the regen process" %
%   N9:29  REGEN_IDLE %
%   N10:0  SYSTEM_STATE  "<datalog> The current state of the system" %
%   N9:1  SYSTEM_PROCESS  "STATE System Process" %
%   N13:2  REGEN_ALARM_BUFFER  "STATE The buffered previous state when the system alarm occured" %
%   N13:3  REGEN_STANDBY_BUFFER  "state The state when the system went to SYSTEM STANDBY" %

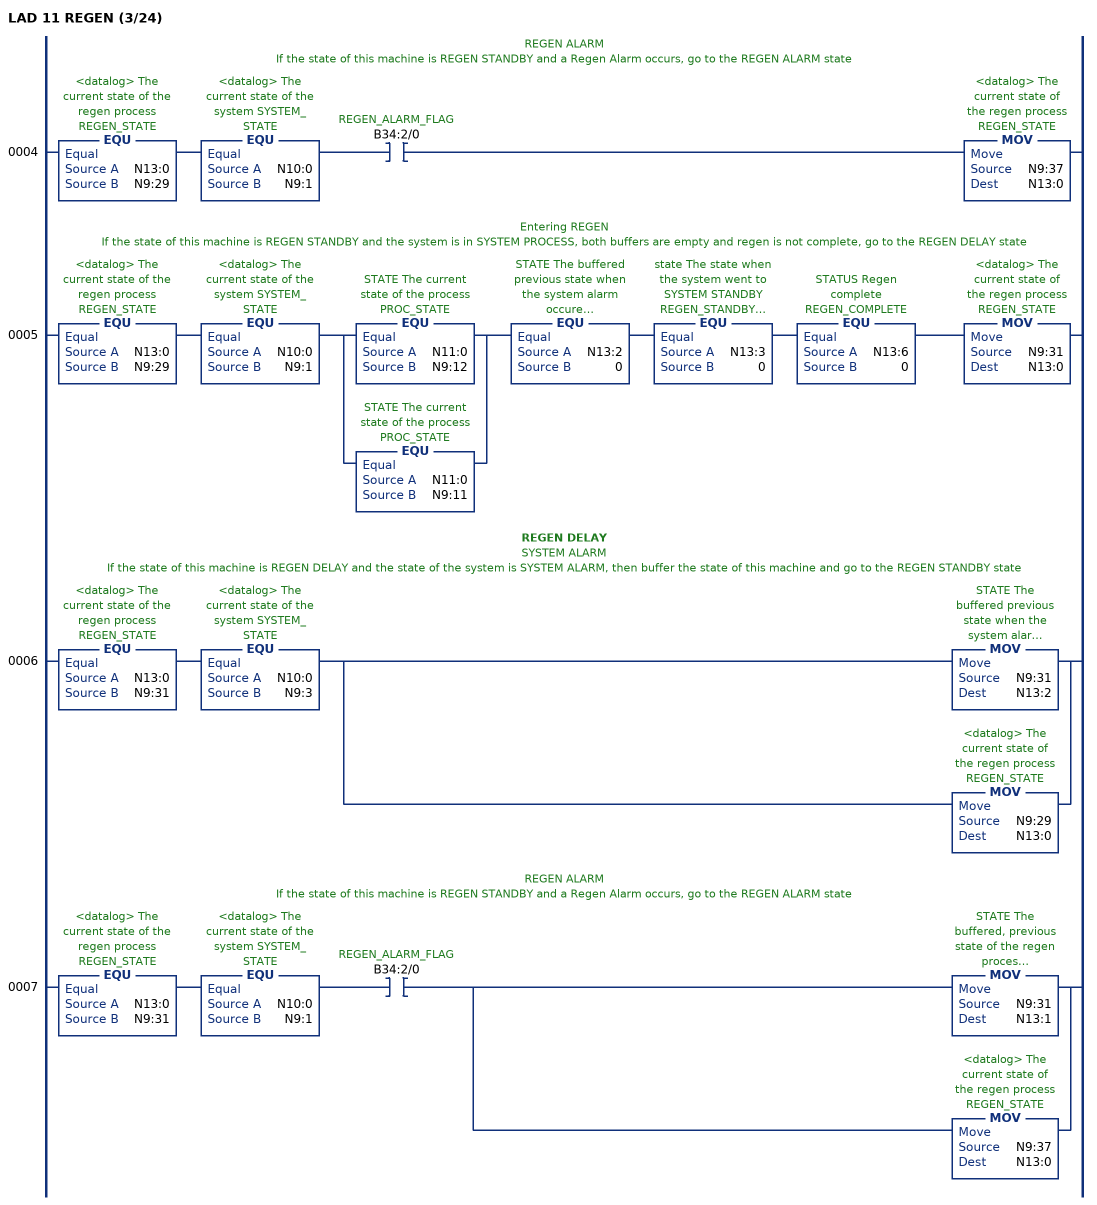
% Rung: 4 %
% REGEN ALARM
% If the state of this machine is REGEN STANDBY and a Regen Alarm occurs, go to the REGEN ALARM state %
SOR EQU N13:0 N9:29 EQU N10:0 N9:1 XIC B34:2/0 MOV N9:37 N13:0 EOR
%   N13:0  REGEN_STATE  "<datalog> The current state of the regen process" %
%   N9:29  REGEN_IDLE %
%   N10:0  SYSTEM_STATE  "<datalog> The current state of the system" %
%   N9:1  SYSTEM_PROCESS  "STATE System Process" %
%   B34:2/0  REGEN_ALARM_FLAG %
%   N9:37  REGEN_ALARM  "STATE Regen Alarm" %
% Rung: 5 %
% Entering REGEN
% If the state of this machine is REGEN STANDBY and the system is in SYSTEM PROCESS, both buffers are empty and regen is not complete, go to the REGEN DELAY state %
SOR EQU N13:0 N9:29 EQU N10:0 N9:1 BST EQU N11:0 N9:12 NXB EQU N11:0 N9:11 BND EQU N13:2 0 EQU N13:3 0 EQU N13:6 0 MOV N9:31 N13:0 EOR
%   N13:0  REGEN_STATE  "<datalog> The current state of the regen process" %
%   N9:29  REGEN_IDLE %
%   N10:0  SYSTEM_STATE  "<datalog> The current state of the system" %
%   N9:1  SYSTEM_PROCESS  "STATE System Process" %
%   N11:0  PROC_STATE  "STATE The current state of the process" %
%   N9:12  PROC_REGEN_A  "STATE Process Purify B" %
%   N9:11  PROC_REGEN_B  "STATE Process Purify A" %
%   N13:2  REGEN_ALARM_BUFFER  "STATE The buffered previous state when the system alarm occured" %
%   N13:3  REGEN_STANDBY_BUFFER  "state The state when the system went to SYSTEM STANDBY" %
%   N13:6  REGEN_COMPLETE  "STATUS Regen complete" %
%   N9:31  REGEN_DELAY  "STATE Regen Delay" %
% Rung: 6 %
% TITLE: REGEN DELAY %
% SYSTEM ALARM
% If the state of this machine is REGEN DELAY and the state of the system is SYSTEM ALARM, then buffer the state of this machine and go to the REGEN STANDBY state %
SOR EQU N13:0 N9:31 EQU N10:0 N9:3 BST MOV N9:31 N13:2 NXB MOV N9:29 N13:0 BND EOR
%   N13:0  REGEN_STATE  "<datalog> The current state of the regen process" %
%   N9:31  REGEN_DELAY  "STATE Regen Delay" %
%   N10:0  SYSTEM_STATE  "<datalog> The current state of the system" %
%   N9:3  SYSTEM_ALARM  "STATE System Alarm" %
%   N13:2  REGEN_ALARM_BUFFER  "STATE The buffered previous state when the system alarm occured" %
%   N9:29  REGEN_IDLE %
% Rung: 7 %
% REGEN ALARM
% If the state of this machine is REGEN STANDBY and a Regen Alarm occurs, go to the REGEN ALARM state %
SOR EQU N13:0 N9:31 EQU N10:0 N9:1 XIC B34:2/0 BST MOV N9:31 N13:1 NXB MOV N9:37 N13:0 BND EOR
%   N13:0  REGEN_STATE  "<datalog> The current state of the regen process" %
%   N9:31  REGEN_DELAY  "STATE Regen Delay" %
%   N10:0  SYSTEM_STATE  "<datalog> The current state of the system" %
%   N9:1  SYSTEM_PROCESS  "STATE System Process" %
%   B34:2/0  REGEN_ALARM_FLAG %
%   N13:1  REGEN_BUFFER  "STATE The buffered, previous state of the regen process" %
%   N9:37  REGEN_ALARM  "STATE Regen Alarm" %

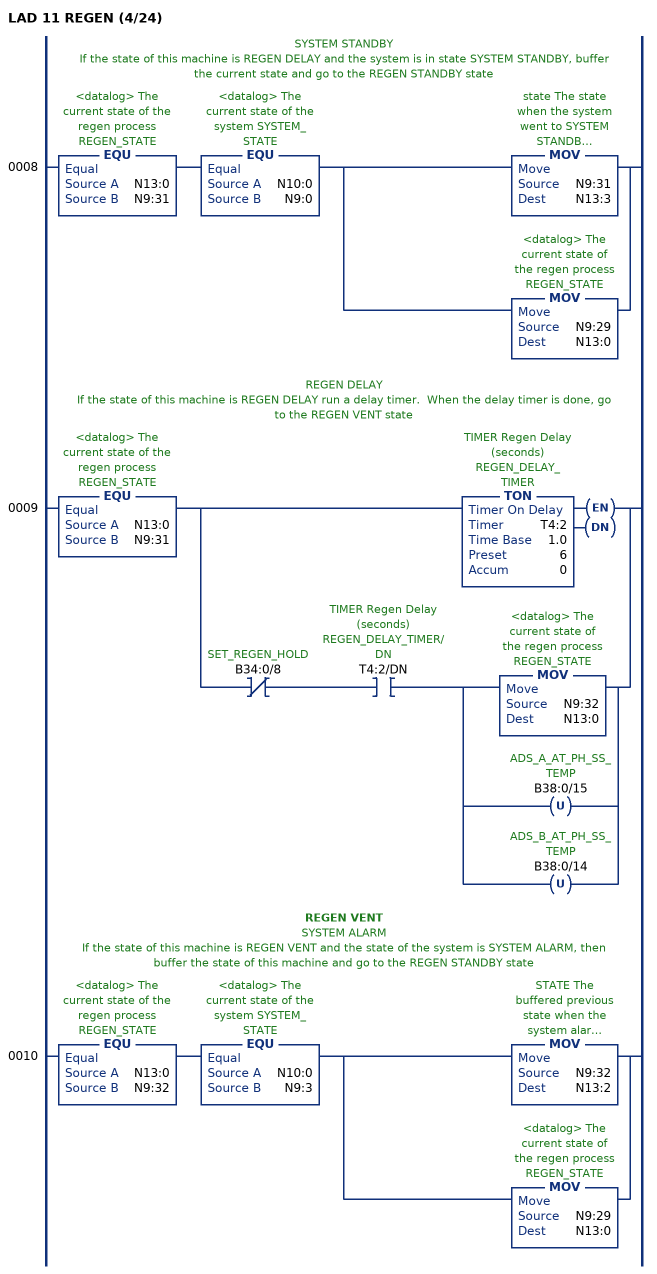
% Rung: 8 %
% SYSTEM STANDBY
% If the state of this machine is REGEN DELAY and the system is in state SYSTEM STANDBY, buffer the current state and go to the REGEN STANDBY state %
SOR EQU N13:0 N9:31 EQU N10:0 N9:0 BST MOV N9:31 N13:3 NXB MOV N9:29 N13:0 BND EOR
%   N13:0  REGEN_STATE  "<datalog> The current state of the regen process" %
%   N9:31  REGEN_DELAY  "STATE Regen Delay" %
%   N10:0  SYSTEM_STATE  "<datalog> The current state of the system" %
%   N9:0  SYSTEM_STANDBY  "STATE System Standby" %
%   N13:3  REGEN_STANDBY_BUFFER  "state The state when the system went to SYSTEM STANDBY" %
%   N9:29  REGEN_IDLE %
% Rung: 9 %
% REGEN DELAY
% If the state of this machine is REGEN DELAY run a delay timer.  When the delay timer is done, go to the REGEN VENT state %
SOR EQU N13:0 N9:31 BST TON T4:2 1.0 6 0 NXB XIO B34:0/8 XIC T4:2/DN BST MOV N9:32 N13:0 NXB OTU B38:0/15 NXB OTU B38:0/14 BND BND EOR
%   N13:0  REGEN_STATE  "<datalog> The current state of the regen process" %
%   N9:31  REGEN_DELAY  "STATE Regen Delay" %
%   T4:2  REGEN_DELAY_TIMER  "TIMER Regen Delay (seconds)" %
%   B34:0/8  SET_REGEN_HOLD %
%   N9:32  REGEN_VENT  "STATE Regen Vent" %
%   B38:0/15  ADS_A_AT_PH_SS_TEMP %
%   B38:0/14  ADS_B_AT_PH_SS_TEMP %
% Rung: 10 %
% TITLE: REGEN VENT %
% SYSTEM ALARM
% If the state of this machine is REGEN VENT and the state of the system is SYSTEM ALARM, then buffer the state of this machine and go to the REGEN STANDBY state %
SOR EQU N13:0 N9:32 EQU N10:0 N9:3 BST MOV N9:32 N13:2 NXB MOV N9:29 N13:0 BND EOR
%   N13:0  REGEN_STATE  "<datalog> The current state of the regen process" %
%   N9:32  REGEN_VENT  "STATE Regen Vent" %
%   N10:0  SYSTEM_STATE  "<datalog> The current state of the system" %
%   N9:3  SYSTEM_ALARM  "STATE System Alarm" %
%   N13:2  REGEN_ALARM_BUFFER  "STATE The buffered previous state when the system alarm occured" %
%   N9:29  REGEN_IDLE %

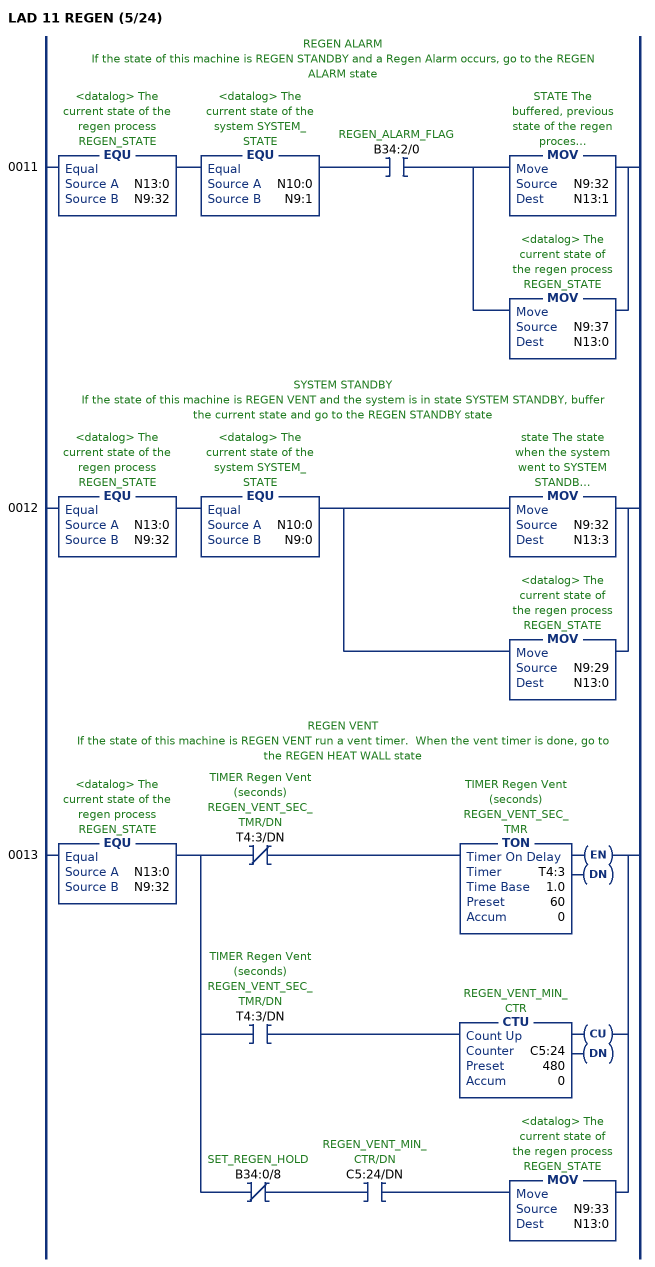
% Rung: 11 %
% REGEN ALARM
% If the state of this machine is REGEN STANDBY and a Regen Alarm occurs, go to the REGEN ALARM state %
SOR EQU N13:0 N9:32 EQU N10:0 N9:1 XIC B34:2/0 BST MOV N9:32 N13:1 NXB MOV N9:37 N13:0 BND EOR
%   N13:0  REGEN_STATE  "<datalog> The current state of the regen process" %
%   N9:32  REGEN_VENT  "STATE Regen Vent" %
%   N10:0  SYSTEM_STATE  "<datalog> The current state of the system" %
%   N9:1  SYSTEM_PROCESS  "STATE System Process" %
%   B34:2/0  REGEN_ALARM_FLAG %
%   N13:1  REGEN_BUFFER  "STATE The buffered, previous state of the regen process" %
%   N9:37  REGEN_ALARM  "STATE Regen Alarm" %
% Rung: 12 %
% SYSTEM STANDBY
% If the state of this machine is REGEN VENT and the system is in state SYSTEM STANDBY, buffer the current state and go to the REGEN STANDBY state %
SOR EQU N13:0 N9:32 EQU N10:0 N9:0 BST MOV N9:32 N13:3 NXB MOV N9:29 N13:0 BND EOR
%   N13:0  REGEN_STATE  "<datalog> The current state of the regen process" %
%   N9:32  REGEN_VENT  "STATE Regen Vent" %
%   N10:0  SYSTEM_STATE  "<datalog> The current state of the system" %
%   N9:0  SYSTEM_STANDBY  "STATE System Standby" %
%   N13:3  REGEN_STANDBY_BUFFER  "state The state when the system went to SYSTEM STANDBY" %
%   N9:29  REGEN_IDLE %
% Rung: 13 %
% REGEN VENT
% If the state of this machine is REGEN VENT run a vent timer.  When the vent timer is done, go to the REGEN HEAT WALL state %
SOR EQU N13:0 N9:32 BST XIO T4:3/DN TON T4:3 1.0 60 0 NXB XIC T4:3/DN CTU C5:24 480 0 NXB XIO B34:0/8 XIC C5:24/DN MOV N9:33 N13:0 BND EOR
%   N13:0  REGEN_STATE  "<datalog> The current state of the regen process" %
%   N9:32  REGEN_VENT  "STATE Regen Vent" %
%   T4:3  REGEN_VENT_SEC_TMR  "TIMER Regen Vent (seconds)" %
%   C5:24  REGEN_VENT_MIN_CTR %
%   B34:0/8  SET_REGEN_HOLD %
%   N9:33  REGEN_HEAT_BED  "STATE Regen Heat wall" %

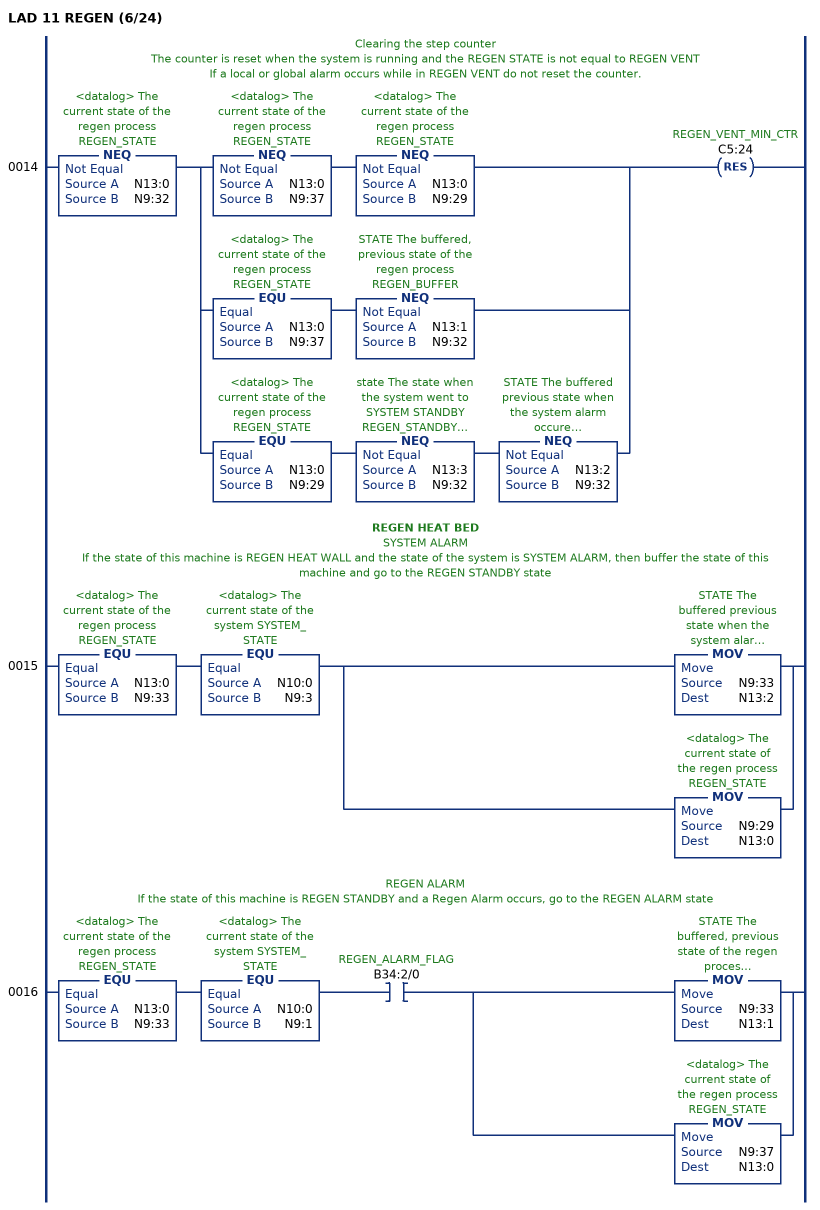
% Rung: 14 %
% Clearing the step counter
% The counter is reset when the system is running and the REGEN STATE is not equal to REGEN VENT
% If a local or global alarm occurs while in REGEN VENT do not reset the counter. %
SOR NEQ N13:0 N9:32 BST NEQ N13:0 N9:37 NEQ N13:0 N9:29 NXB EQU N13:0 N9:37 NEQ N13:1 N9:32 NXB EQU N13:0 N9:29 NEQ N13:3 N9:32 NEQ N13:2 N9:32 BND RES C5:24 EOR
%   N13:0  REGEN_STATE  "<datalog> The current state of the regen process" %
%   N9:32  REGEN_VENT  "STATE Regen Vent" %
%   N9:37  REGEN_ALARM  "STATE Regen Alarm" %
%   N9:29  REGEN_IDLE %
%   N13:1  REGEN_BUFFER  "STATE The buffered, previous state of the regen process" %
%   N13:3  REGEN_STANDBY_BUFFER  "state The state when the system went to SYSTEM STANDBY" %
%   N13:2  REGEN_ALARM_BUFFER  "STATE The buffered previous state when the system alarm occured" %
%   C5:24  REGEN_VENT_MIN_CTR %
% Rung: 15 %
% TITLE: REGEN HEAT BED %
% SYSTEM ALARM
% If the state of this machine is REGEN HEAT WALL and the state of the system is SYSTEM ALARM, then buffer the state of this machine and go to the REGEN STANDBY state %
SOR EQU N13:0 N9:33 EQU N10:0 N9:3 BST MOV N9:33 N13:2 NXB MOV N9:29 N13:0 BND EOR
%   N13:0  REGEN_STATE  "<datalog> The current state of the regen process" %
%   N9:33  REGEN_HEAT_BED  "STATE Regen Heat wall" %
%   N10:0  SYSTEM_STATE  "<datalog> The current state of the system" %
%   N9:3  SYSTEM_ALARM  "STATE System Alarm" %
%   N13:2  REGEN_ALARM_BUFFER  "STATE The buffered previous state when the system alarm occured" %
%   N9:29  REGEN_IDLE %
% Rung: 16 %
% REGEN ALARM
% If the state of this machine is REGEN STANDBY and a Regen Alarm occurs, go to the REGEN ALARM state %
SOR EQU N13:0 N9:33 EQU N10:0 N9:1 XIC B34:2/0 BST MOV N9:33 N13:1 NXB MOV N9:37 N13:0 BND EOR
%   N13:0  REGEN_STATE  "<datalog> The current state of the regen process" %
%   N9:33  REGEN_HEAT_BED  "STATE Regen Heat wall" %
%   N10:0  SYSTEM_STATE  "<datalog> The current state of the system" %
%   N9:1  SYSTEM_PROCESS  "STATE System Process" %
%   B34:2/0  REGEN_ALARM_FLAG %
%   N13:1  REGEN_BUFFER  "STATE The buffered, previous state of the regen process" %
%   N9:37  REGEN_ALARM  "STATE Regen Alarm" %

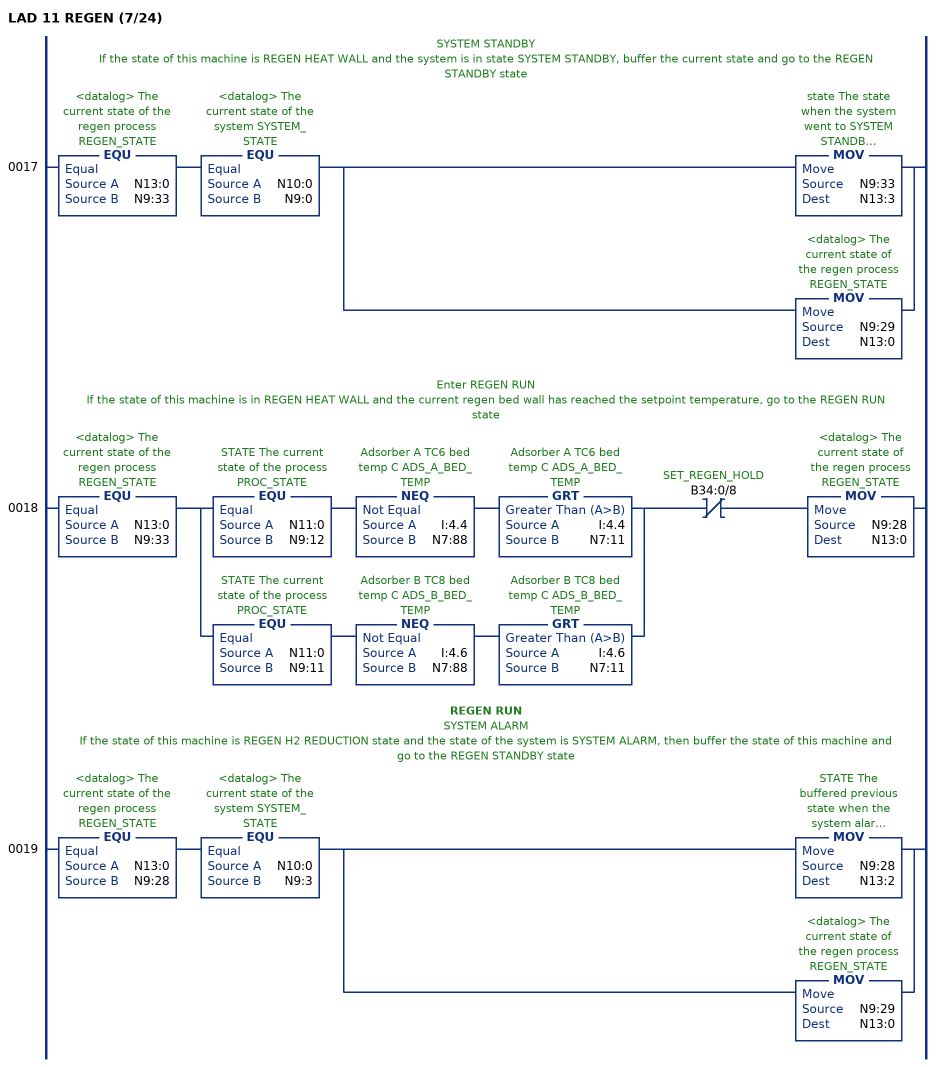
% Rung: 17 %
% SYSTEM STANDBY
% If the state of this machine is REGEN HEAT WALL and the system is in state SYSTEM STANDBY, buffer the current state and go to the REGEN STANDBY state %
SOR EQU N13:0 N9:33 EQU N10:0 N9:0 BST MOV N9:33 N13:3 NXB MOV N9:29 N13:0 BND EOR
%   N13:0  REGEN_STATE  "<datalog> The current state of the regen process" %
%   N9:33  REGEN_HEAT_BED  "STATE Regen Heat wall" %
%   N10:0  SYSTEM_STATE  "<datalog> The current state of the system" %
%   N9:0  SYSTEM_STANDBY  "STATE System Standby" %
%   N13:3  REGEN_STANDBY_BUFFER  "state The state when the system went to SYSTEM STANDBY" %
%   N9:29  REGEN_IDLE %
% Rung: 18 %
% Enter REGEN RUN
% If the state of this machine is in REGEN HEAT WALL and the current regen bed wall has reached the setpoint temperature, go to the REGEN RUN state %
SOR EQU N13:0 N9:33 BST EQU N11:0 N9:12 NEQ I:4.4 N7:88 GRT I:4.4 N7:11 NXB EQU N11:0 N9:11 NEQ I:4.6 N7:88 GRT I:4.6 N7:11 BND XIO B34:0/8 MOV N9:28 N13:0 EOR
%   N13:0  REGEN_STATE  "<datalog> The current state of the regen process" %
%   N9:33  REGEN_HEAT_BED  "STATE Regen Heat wall" %
%   N11:0  PROC_STATE  "STATE The current state of the process" %
%   N9:12  PROC_REGEN_A  "STATE Process Purify B" %
%   I:4.4  ADS_A_BED_TEMP  "Adsorber A TC6 bed temp C" %
%   N7:88  TC_OPEN_SP  "CONFIG The value read by an open TC input" %
%   N7:11  ADS_BED_TEMP_HIGH  "CONFIG The temp at which the regen process may continue" %
%   N9:11  PROC_REGEN_B  "STATE Process Purify A" %
%   I:4.6  ADS_B_BED_TEMP  "Adsorber B TC8 bed temp C" %
%   B34:0/8  SET_REGEN_HOLD %
%   N9:28  REGEN_RUN %
% Rung: 19 %
% TITLE: REGEN RUN %
% SYSTEM ALARM
% If the state of this machine is REGEN H2 REDUCTION state and the state of the system is SYSTEM ALARM, then buffer the state of this machine and go to the REGEN STANDBY state %
SOR EQU N13:0 N9:28 EQU N10:0 N9:3 BST MOV N9:28 N13:2 NXB MOV N9:29 N13:0 BND EOR
%   N13:0  REGEN_STATE  "<datalog> The current state of the regen process" %
%   N9:28  REGEN_RUN %
%   N10:0  SYSTEM_STATE  "<datalog> The current state of the system" %
%   N9:3  SYSTEM_ALARM  "STATE System Alarm" %
%   N13:2  REGEN_ALARM_BUFFER  "STATE The buffered previous state when the system alarm occured" %
%   N9:29  REGEN_IDLE %

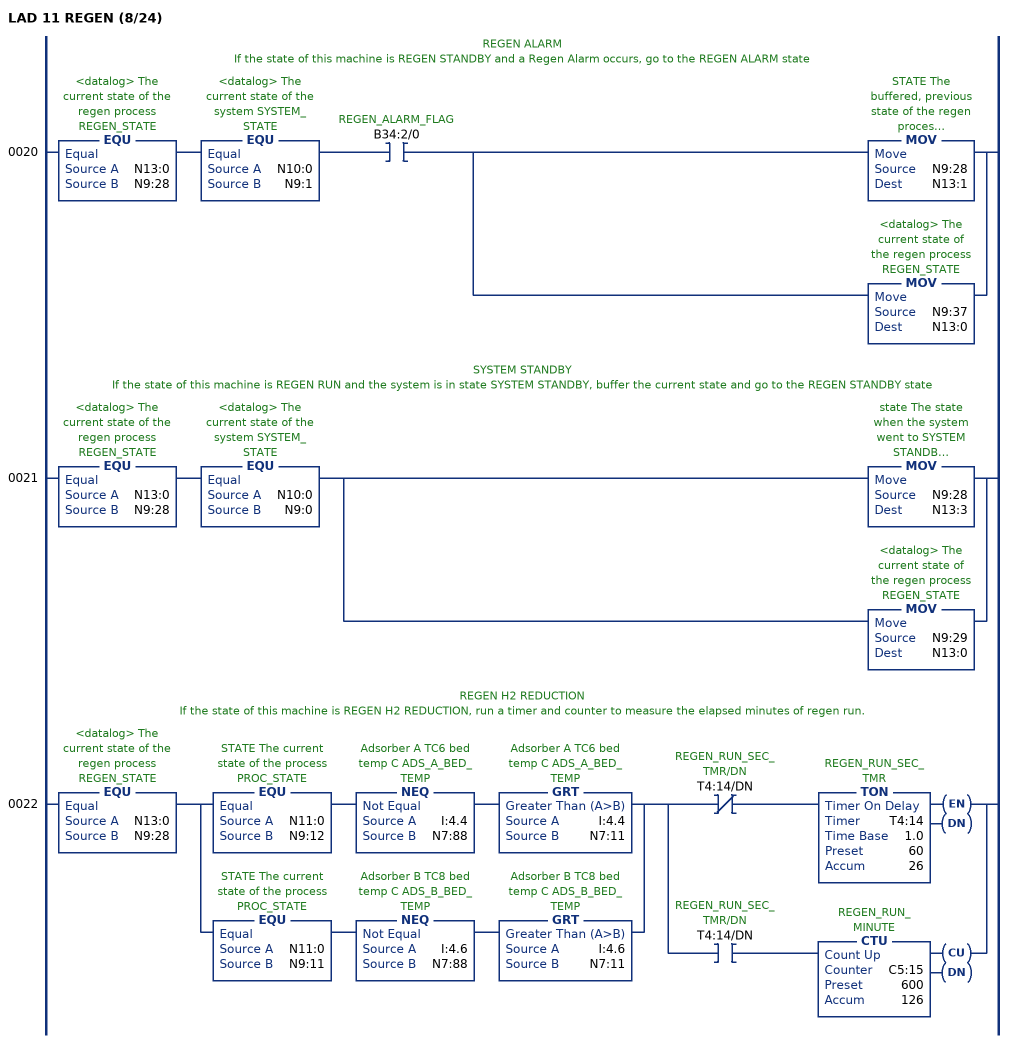
% Rung: 20 %
% REGEN ALARM
% If the state of this machine is REGEN STANDBY and a Regen Alarm occurs, go to the REGEN ALARM state %
SOR EQU N13:0 N9:28 EQU N10:0 N9:1 XIC B34:2/0 BST MOV N9:28 N13:1 NXB MOV N9:37 N13:0 BND EOR
%   N13:0  REGEN_STATE  "<datalog> The current state of the regen process" %
%   N9:28  REGEN_RUN %
%   N10:0  SYSTEM_STATE  "<datalog> The current state of the system" %
%   N9:1  SYSTEM_PROCESS  "STATE System Process" %
%   B34:2/0  REGEN_ALARM_FLAG %
%   N13:1  REGEN_BUFFER  "STATE The buffered, previous state of the regen process" %
%   N9:37  REGEN_ALARM  "STATE Regen Alarm" %
% Rung: 21 %
% SYSTEM STANDBY
% If the state of this machine is REGEN RUN and the system is in state SYSTEM STANDBY, buffer the current state and go to the REGEN STANDBY state %
SOR EQU N13:0 N9:28 EQU N10:0 N9:0 BST MOV N9:28 N13:3 NXB MOV N9:29 N13:0 BND EOR
%   N13:0  REGEN_STATE  "<datalog> The current state of the regen process" %
%   N9:28  REGEN_RUN %
%   N10:0  SYSTEM_STATE  "<datalog> The current state of the system" %
%   N9:0  SYSTEM_STANDBY  "STATE System Standby" %
%   N13:3  REGEN_STANDBY_BUFFER  "state The state when the system went to SYSTEM STANDBY" %
%   N9:29  REGEN_IDLE %
% Rung: 22 %
% REGEN H2 REDUCTION
% If the state of this machine is REGEN H2 REDUCTION, run a timer and counter to measure the elapsed minutes of regen run. %
SOR EQU N13:0 N9:28 BST EQU N11:0 N9:12 NEQ I:4.4 N7:88 GRT I:4.4 N7:11 NXB EQU N11:0 N9:11 NEQ I:4.6 N7:88 GRT I:4.6 N7:11 BND BST XIO T4:14/DN TON T4:14 1.0 60 26 NXB XIC T4:14/DN CTU C5:15 600 126 BND EOR
%   N13:0  REGEN_STATE  "<datalog> The current state of the regen process" %
%   N9:28  REGEN_RUN %
%   N11:0  PROC_STATE  "STATE The current state of the process" %
%   N9:12  PROC_REGEN_A  "STATE Process Purify B" %
%   I:4.4  ADS_A_BED_TEMP  "Adsorber A TC6 bed temp C" %
%   N7:88  TC_OPEN_SP  "CONFIG The value read by an open TC input" %
%   N7:11  ADS_BED_TEMP_HIGH  "CONFIG The temp at which the regen process may continue" %
%   N9:11  PROC_REGEN_B  "STATE Process Purify A" %
%   I:4.6  ADS_B_BED_TEMP  "Adsorber B TC8 bed temp C" %
%   T4:14  REGEN_RUN_SEC_TMR %
%   C5:15  REGEN_RUN_MINUTE %

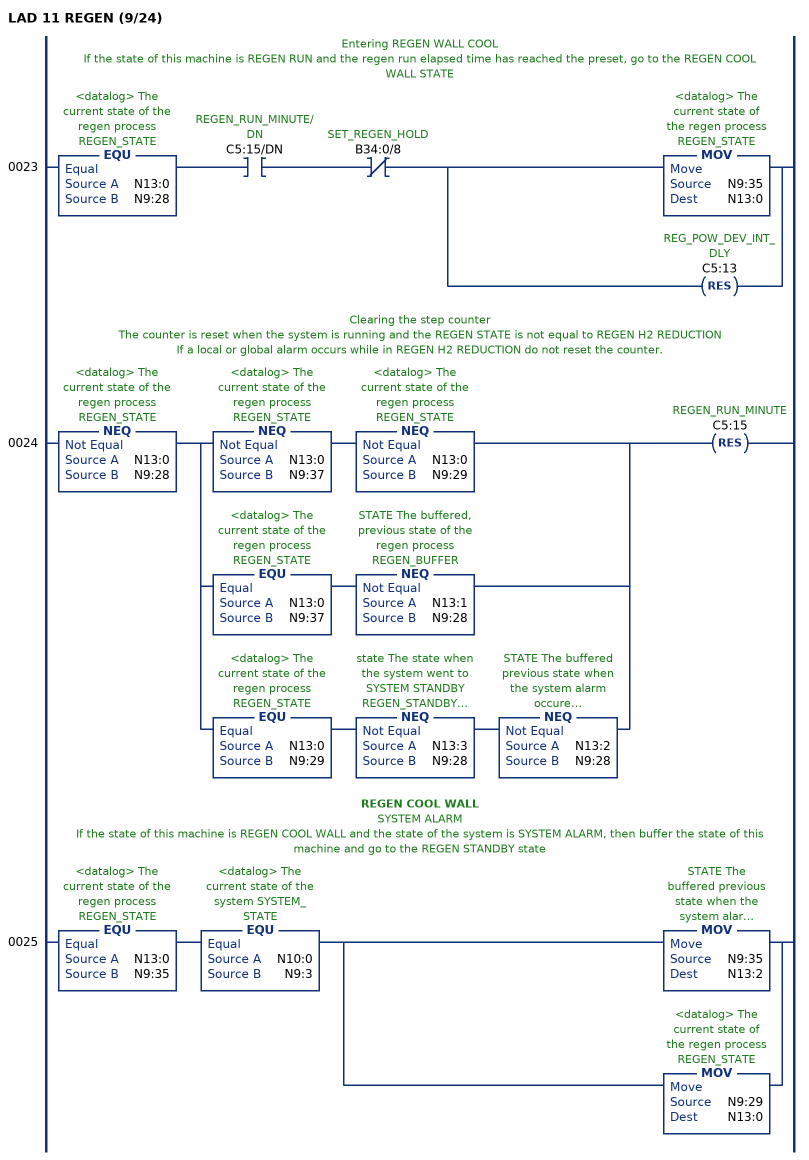
% Rung: 23 %
% Entering REGEN WALL COOL
% If the state of this machine is REGEN RUN and the regen run elapsed time has reached the preset, go to the REGEN COOL WALL STATE %
SOR EQU N13:0 N9:28 XIC C5:15/DN XIO B34:0/8 BST MOV N9:35 N13:0 NXB RES C5:13 BND EOR
%   N13:0  REGEN_STATE  "<datalog> The current state of the regen process" %
%   N9:28  REGEN_RUN %
%   C5:15  REGEN_RUN_MINUTE %
%   B34:0/8  SET_REGEN_HOLD %
%   N9:35  REGEN_COOL_WALL  "STATE Regen Cool wall" %
%   C5:13  REG_POW_DEV_INT_DLY %
% Rung: 24 %
% Clearing the step counter
% The counter is reset when the system is running and the REGEN STATE is not equal to REGEN H2 REDUCTION
% If a local or global alarm occurs while in REGEN H2 REDUCTION do not reset the counter. %
SOR NEQ N13:0 N9:28 BST NEQ N13:0 N9:37 NEQ N13:0 N9:29 NXB EQU N13:0 N9:37 NEQ N13:1 N9:28 NXB EQU N13:0 N9:29 NEQ N13:3 N9:28 NEQ N13:2 N9:28 BND RES C5:15 EOR
%   N13:0  REGEN_STATE  "<datalog> The current state of the regen process" %
%   N9:28  REGEN_RUN %
%   N9:37  REGEN_ALARM  "STATE Regen Alarm" %
%   N9:29  REGEN_IDLE %
%   N13:1  REGEN_BUFFER  "STATE The buffered, previous state of the regen process" %
%   N13:3  REGEN_STANDBY_BUFFER  "state The state when the system went to SYSTEM STANDBY" %
%   N13:2  REGEN_ALARM_BUFFER  "STATE The buffered previous state when the system alarm occured" %
%   C5:15  REGEN_RUN_MINUTE %
% Rung: 25 %
% TITLE: REGEN COOL WALL %
% SYSTEM ALARM
% If the state of this machine is REGEN COOL WALL and the state of the system is SYSTEM ALARM, then buffer the state of this machine and go to the REGEN STANDBY state %
SOR EQU N13:0 N9:35 EQU N10:0 N9:3 BST MOV N9:35 N13:2 NXB MOV N9:29 N13:0 BND EOR
%   N13:0  REGEN_STATE  "<datalog> The current state of the regen process" %
%   N9:35  REGEN_COOL_WALL  "STATE Regen Cool wall" %
%   N10:0  SYSTEM_STATE  "<datalog> The current state of the system" %
%   N9:3  SYSTEM_ALARM  "STATE System Alarm" %
%   N13:2  REGEN_ALARM_BUFFER  "STATE The buffered previous state when the system alarm occured" %
%   N9:29  REGEN_IDLE %

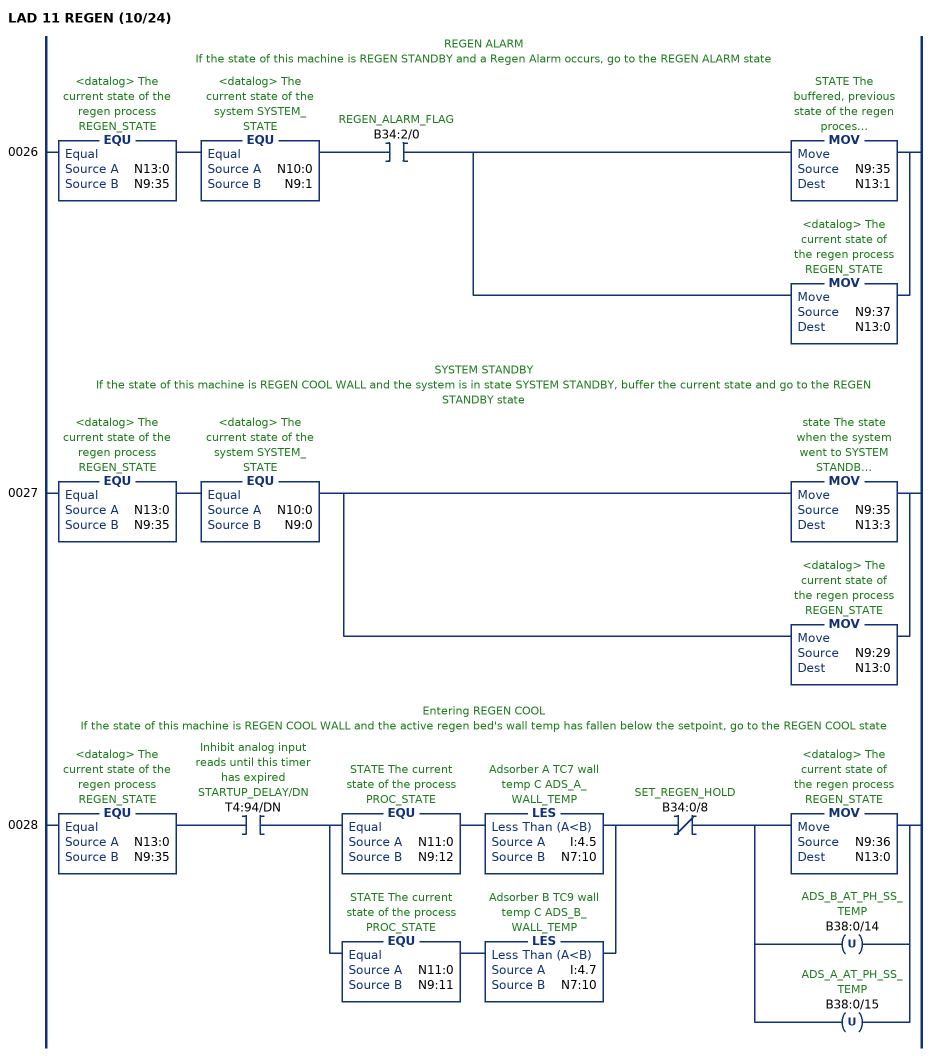
% Rung: 26 %
% REGEN ALARM
% If the state of this machine is REGEN STANDBY and a Regen Alarm occurs, go to the REGEN ALARM state %
SOR EQU N13:0 N9:35 EQU N10:0 N9:1 XIC B34:2/0 BST MOV N9:35 N13:1 NXB MOV N9:37 N13:0 BND EOR
%   N13:0  REGEN_STATE  "<datalog> The current state of the regen process" %
%   N9:35  REGEN_COOL_WALL  "STATE Regen Cool wall" %
%   N10:0  SYSTEM_STATE  "<datalog> The current state of the system" %
%   N9:1  SYSTEM_PROCESS  "STATE System Process" %
%   B34:2/0  REGEN_ALARM_FLAG %
%   N13:1  REGEN_BUFFER  "STATE The buffered, previous state of the regen process" %
%   N9:37  REGEN_ALARM  "STATE Regen Alarm" %
% Rung: 27 %
% SYSTEM STANDBY
% If the state of this machine is REGEN COOL WALL and the system is in state SYSTEM STANDBY, buffer the current state and go to the REGEN STANDBY state %
SOR EQU N13:0 N9:35 EQU N10:0 N9:0 BST MOV N9:35 N13:3 NXB MOV N9:29 N13:0 BND EOR
%   N13:0  REGEN_STATE  "<datalog> The current state of the regen process" %
%   N9:35  REGEN_COOL_WALL  "STATE Regen Cool wall" %
%   N10:0  SYSTEM_STATE  "<datalog> The current state of the system" %
%   N9:0  SYSTEM_STANDBY  "STATE System Standby" %
%   N13:3  REGEN_STANDBY_BUFFER  "state The state when the system went to SYSTEM STANDBY" %
%   N9:29  REGEN_IDLE %
% Rung: 28 %
% Entering REGEN COOL
% If the state of this machine is REGEN COOL WALL and the active regen bed's wall temp has fallen below the setpoint, go to the REGEN COOL state %
SOR EQU N13:0 N9:35 XIC T4:94/DN BST EQU N11:0 N9:12 LES I:4.5 N7:10 NXB EQU N11:0 N9:11 LES I:4.7 N7:10 BND XIO B34:0/8 BST MOV N9:36 N13:0 NXB OTU B38:0/14 NXB OTU B38:0/15 BND EOR
%   N13:0  REGEN_STATE  "<datalog> The current state of the regen process" %
%   N9:35  REGEN_COOL_WALL  "STATE Regen Cool wall" %
%   T4:94  STARTUP_DELAY  "Inhibit analog input reads until this timer has expired" %
%   N11:0  PROC_STATE  "STATE The current state of the process" %
%   N9:12  PROC_REGEN_A  "STATE Process Purify B" %
%   I:4.5  ADS_A_WALL_TEMP  "Adsorber A TC7 wall temp C" %
%   N7:10  ADS_WALL_TEMP_COOL  "CONFIG The temp at which the adsorber wall is deemed to be cool enough to purify" %
%   N9:11  PROC_REGEN_B  "STATE Process Purify A" %
%   I:4.7  ADS_B_WALL_TEMP  "Adsorber B TC9 wall temp C" %
%   B34:0/8  SET_REGEN_HOLD %
%   N9:36  REGEN_COOL  "STATE Regen Cool" %
%   B38:0/14  ADS_B_AT_PH_SS_TEMP %
%   B38:0/15  ADS_A_AT_PH_SS_TEMP %

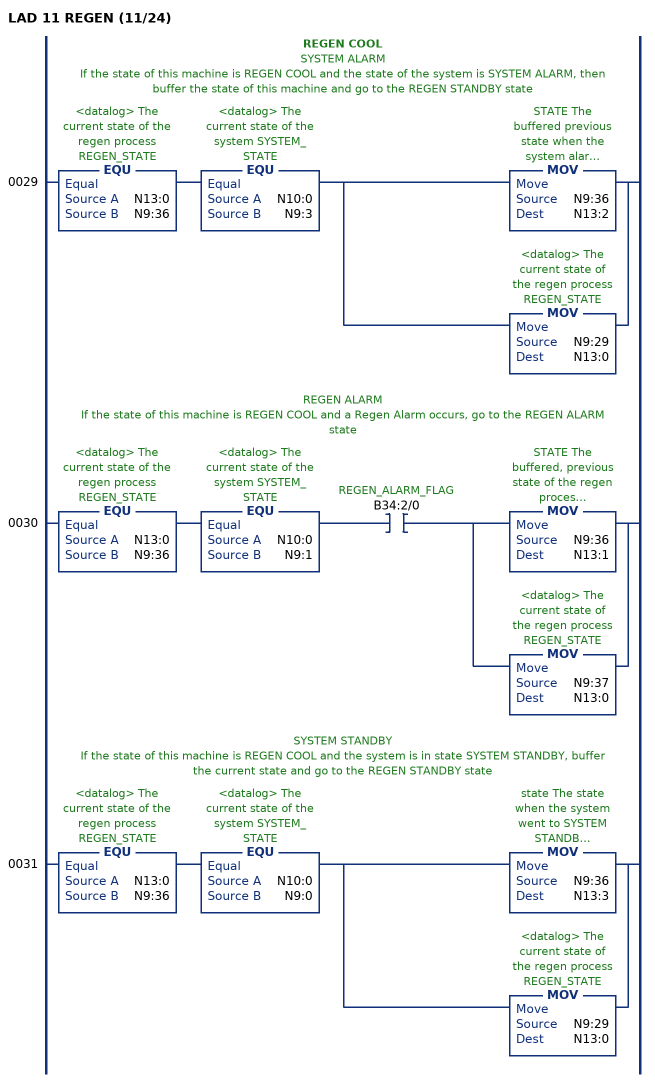
% Rung: 29 %
% TITLE: REGEN COOL %
% SYSTEM ALARM
% If the state of this machine is REGEN COOL and the state of the system is SYSTEM ALARM, then buffer the state of this machine and go to the REGEN STANDBY state %
SOR EQU N13:0 N9:36 EQU N10:0 N9:3 BST MOV N9:36 N13:2 NXB MOV N9:29 N13:0 BND EOR
%   N13:0  REGEN_STATE  "<datalog> The current state of the regen process" %
%   N9:36  REGEN_COOL  "STATE Regen Cool" %
%   N10:0  SYSTEM_STATE  "<datalog> The current state of the system" %
%   N9:3  SYSTEM_ALARM  "STATE System Alarm" %
%   N13:2  REGEN_ALARM_BUFFER  "STATE The buffered previous state when the system alarm occured" %
%   N9:29  REGEN_IDLE %
% Rung: 30 %
% REGEN ALARM
% If the state of this machine is REGEN COOL and a Regen Alarm occurs, go to the REGEN ALARM state %
SOR EQU N13:0 N9:36 EQU N10:0 N9:1 XIC B34:2/0 BST MOV N9:36 N13:1 NXB MOV N9:37 N13:0 BND EOR
%   N13:0  REGEN_STATE  "<datalog> The current state of the regen process" %
%   N9:36  REGEN_COOL  "STATE Regen Cool" %
%   N10:0  SYSTEM_STATE  "<datalog> The current state of the system" %
%   N9:1  SYSTEM_PROCESS  "STATE System Process" %
%   B34:2/0  REGEN_ALARM_FLAG %
%   N13:1  REGEN_BUFFER  "STATE The buffered, previous state of the regen process" %
%   N9:37  REGEN_ALARM  "STATE Regen Alarm" %
% Rung: 31 %
% SYSTEM STANDBY
% If the state of this machine is REGEN COOL and the system is in state SYSTEM STANDBY, buffer the current state and go to the REGEN STANDBY state %
SOR EQU N13:0 N9:36 EQU N10:0 N9:0 BST MOV N9:36 N13:3 NXB MOV N9:29 N13:0 BND EOR
%   N13:0  REGEN_STATE  "<datalog> The current state of the regen process" %
%   N9:36  REGEN_COOL  "STATE Regen Cool" %
%   N10:0  SYSTEM_STATE  "<datalog> The current state of the system" %
%   N9:0  SYSTEM_STANDBY  "STATE System Standby" %
%   N13:3  REGEN_STANDBY_BUFFER  "state The state when the system went to SYSTEM STANDBY" %
%   N9:29  REGEN_IDLE %

